C05461=1057.232,60.165,424.870,171.464,30.590,155.709
C05462=1057.237,60.415,424.853,171.466,30.593,155.709
C05463=1057.243,60.664,424.836,171.467,30.594,155.710
C05464=1057.249,60.914,424.818,171.468,30.597,155.710
C05465=1057.256,61.162,424.801,171.470,30.599,155.710
C05466=1057.263,61.412,424.784,171.472,30.602,155.711
C05467=1057.269,61.697,424.764,171.474,30.605,155.711
C05468=1057.277,61.982,424.744,171.476,30.607,155.712
C05469=1057.283,62.267,424.724,171.477,30.610,155.712
C05470=1057.291,62.551,424.705,171.479,30.613,155.712
C05471=1057.297,62.801,424.687,171.480,30.615,155.713
C05472=1057.303,63.051,424.671,171.482,30.618,155.713
C05473=1057.309,63.300,424.653,171.484,30.620,155.713
C05474=1057.316,63.550,424.635,171.485,30.622,155.714
C05475=1057.321,63.799,424.618,171.486,30.624,155.714
C05476=1057.328,64.048,424.600,171.488,30.627,155.714
C05477=1057.334,64.297,424.583,171.490,30.629,155.715
C05478=1057.341,64.547,424.565,171.491,30.632,155.715
C05479=1057.346,64.796,424.548,171.493,30.634,155.715
C05480=1057.352,65.045,424.530,171.494,30.636,155.716
C05481=1057.358,65.294,424.513,171.496,30.639,155.716
C05482=1057.365,65.544,424.495,171.497,30.641,155.717
C05483=1057.370,65.793,424.478,171.499,30.644,155.717
C05484=1057.377,66.042,424.460,171.500,30.647,155.717
C05485=1057.382,66.291,424.443,171.501,30.649,155.718
C05486=1057.389,66.541,424.425,171.503,30.651,155.718
C05487=1057.395,66.790,424.408,171.505,30.653,155.718
C05488=1057.401,67.040,424.390,171.507,30.656,155.719
C05489=1057.406,67.289,424.372,171.508,30.659,155.719
C05490=1057.413,67.538,424.355,171.509,30.661,155.720
C05491=1057.419,67.788,424.337,171.511,30.663,155.720
C05492=1057.425,68.037,424.319,171.512,30.666,155.720
C05493=1057.431,68.287,424.301,171.514,30.668,155.721
C05494=1057.437,68.535,424.284,171.516,30.671,155.721
C05495=1057.443,68.785,424.267,171.517,30.673,155.721
C05496=1057.449,69.034,424.249,171.518,30.675,155.722
C05497=1057.455,69.284,424.231,171.520,30.678,155.722
C05498=1057.461,69.533,424.214,171.522,30.680,155.722
C05499=1057.467,69.782,424.196,171.524,30.683,155.723
C05500=1057.474,70.031,424.177,171.524,30.685,155.723
C05501=1057.479,70.280,424.160,171.526,30.688,155.724
C05502=1057.486,70.530,424.142,171.528,30.690,155.724
C05503=1057.492,70.779,424.125,171.529,30.693,155.724
C05504=1057.498,71.029,424.107,171.531,30.695,155.725
C05505=1057.503,71.278,424.089,171.532,30.698,155.725
C05506=1057.510,71.527,424.072,171.534,30.700,155.726
C05507=1057.516,71.777,424.053,171.535,30.702,155.726
C05508=1057.522,72.026,424.035,171.537,30.705,155.726
C05509=1057.528,72.275,424.018,171.539,30.708,155.727
C05510=1057.534,72.524,424.000,171.540,30.710,155.727
C05511=1057.540,72.774,423.983,171.541,30.712,155.727
C05512=1057.546,73.023,423.964,171.543,30.715,155.728
C05513=1057.552,73.272,423.946,171.545,30.717,155.728
C05514=1057.558,73.522,423.928,171.546,30.720,155.728
C05515=1057.564,73.771,423.911,171.548,30.722,155.729
C05516=1057.570,74.020,423.892,171.549,30.725,155.729
C05517=1057.576,74.270,423.874,171.550,30.727,155.730
C05518=1057.582,74.519,423.857,171.552,30.730,155.730
C05519=1057.589,74.768,423.839,171.554,30.732,155.730
C05520=1057.594,75.017,423.821,171.556,30.735,155.731
C05521=1057.600,75.266,423.803,171.556,30.737,155.731
C05522=1057.607,75.516,423.785,171.558,30.739,155.731
C05523=1057.612,75.764,423.767,171.560,30.742,155.732
C05524=1057.619,76.014,423.749,171.561,30.744,155.732
C05525=1057.625,76.264,423.731,171.563,30.747,155.733
C05526=1057.630,76.512,423.713,171.564,30.749,155.733
C05527=1057.637,76.762,423.695,171.566,30.752,155.733
C05528=1057.643,77.012,423.677,171.567,30.754,155.734
C05529=1057.649,77.260,423.659,171.569,30.757,155.734
C05530=1057.655,77.510,423.641,171.571,30.759,155.734
C05531=1057.662,77.795,423.620,171.572,30.762,155.735
C05532=1057.669,78.080,423.600,171.574,30.765,155.735
C05533=1057.676,78.364,423.579,171.576,30.767,155.736
C05534=1057.683,78.649,423.558,171.578,30.771,155.736
C05535=1057.689,78.899,423.540,171.579,30.773,155.737
C05536=1057.695,79.147,423.522,171.580,30.775,155.737
C05537=1057.700,79.397,423.503,171.582,30.778,155.737
C05538=1057.706,79.647,423.485,171.584,30.781,155.738
C05539=1057.712,79.896,423.467,171.585,30.783,155.738
C05540=1057.718,80.145,423.449,171.587,30.785,155.738
C05541=1057.725,80.394,423.430,171.588,30.788,155.739
C05542=1057.730,80.643,423.413,171.589,30.791,155.739
C05543=1057.736,80.893,423.394,171.591,30.793,155.740
C05544=1057.742,81.143,423.376,171.593,30.795,155.740
C05545=1057.748,81.391,423.357,171.595,30.798,155.740
C05546=1057.754,81.641,423.339,171.596,30.801,155.741
C05547=1057.760,81.890,423.321,171.597,30.803,155.741
C05548=1057.766,82.139,423.303,171.599,30.805,155.742
C05549=1057.772,82.388,423.284,171.601,30.808,155.742
C05550=1057.778,82.638,423.265,171.602,30.811,155.742
C05551=1057.784,82.887,423.247,171.604,30.813,155.743
C05552=1057.790,83.136,423.229,171.605,30.815,155.743
C05553=1057.796,83.385,423.211,171.606,30.818,155.744
C05554=1057.802,83.635,423.193,171.608,30.821,155.744
C05555=1057.808,83.885,423.174,171.610,30.823,155.744
C05556=1057.814,84.133,423.156,171.612,30.825,155.745
C05557=1057.820,84.382,423.137,171.613,30.828,155.745
C05558=1057.826,84.632,423.119,171.614,30.830,155.745
C05559=1057.833,84.881,423.101,171.616,30.833,155.746
C05560=1057.837,85.130,423.082,171.618,30.835,155.746
C05561=1057.844,85.379,423.064,171.619,30.838,155.747
C05562=1057.850,85.629,423.045,171.621,30.840,155.747
C05563=1057.856,85.878,423.027,171.622,30.843,155.747
C05564=1057.862,86.127,423.009,171.623,30.845,155.748
C05565=1057.868,86.376,422.990,171.625,30.847,155.748
C05566=1057.874,86.626,422.972,171.627,30.850,155.748
C05567=1057.880,86.875,422.953,171.629,30.853,155.749
C05568=1057.887,87.124,422.934,171.630,30.855,155.749
C05569=1057.892,87.373,422.917,171.631,30.857,155.750
C05570=1057.898,87.623,422.898,171.633,30.860,155.750
C05571=1057.905,87.872,422.879,171.635,30.863,155.750
C05572=1057.911,88.121,422.860,171.636,30.865,155.751
C05573=1057.917,88.371,422.842,171.638,30.867,155.751
C05574=1057.923,88.619,422.824,171.639,30.870,155.752
C05575=1057.929,88.868,422.805,171.641,30.872,155.752
C05576=1057.935,89.118,422.786,171.642,30.875,155.752
C05577=1057.941,89.367,422.768,171.644,30.877,155.753
C05578=1057.948,89.616,422.750,171.646,30.880,155.753
C05579=1057.953,89.866,422.730,171.648,30.882,155.753
C05580=1057.960,90.115,422.712,171.648,30.885,155.754
C05581=1057.965,90.364,422.694,171.650,30.887,155.754
C05582=1057.972,90.613,422.675,171.652,30.890,155.754
C05583=1057.977,90.863,422.656,171.654,30.892,155.755
C05584=1057.984,91.112,422.638,171.655,30.895,155.755
C05585=1057.989,91.361,422.618,171.656,30.897,155.756
C05586=1057.996,91.610,422.600,171.658,30.900,155.756
C05587=1058.001,91.860,422.582,171.659,30.902,155.756
C05588=1058.007,92.109,422.563,171.661,30.905,155.757
C05589=1058.013,92.358,422.544,171.663,30.907,155.757
C05590=1058.019,92.607,422.525,171.665,30.910,155.758
C05591=1058.025,92.857,422.506,171.665,30.912,155.758
C05592=1058.031,93.106,422.487,171.667,30.915,155.758
C05593=1058.036,93.355,422.468,171.669,30.917,155.759
C05594=1058.043,93.604,422.450,171.671,30.920,155.759
C05595=1058.049,93.889,422.428,171.673,30.923,155.760
C05596=1058.057,94.174,422.407,171.674,30.926,155.760
C05597=1058.063,94.458,422.385,171.676,30.929,155.761
C05598=1058.070,94.743,422.363,171.678,30.931,155.761
C05599=1058.076,94.992,422.345,171.679,30.934,155.761
C05600=1058.082,95.242,422.325,171.681,30.937,155.762
C05601=1058.089,95.491,422.307,171.682,30.939,155.762
C05602=1058.094,95.740,422.288,171.684,30.941,155.763
C05603=1058.101,95.990,422.269,171.685,30.944,155.763
C05604=1058.106,96.239,422.250,171.687,30.947,155.763
C05605=1058.112,96.487,422.231,171.689,30.949,155.764
C05606=1058.118,96.737,422.212,171.691,30.951,155.764
C05607=1058.124,96.986,422.194,171.691,30.954,155.764
C05608=1058.130,97.235,422.174,171.693,30.957,155.765
C05609=1058.136,97.484,422.156,171.695,30.959,155.765
C05610=1058.142,97.734,422.136,171.697,30.961,155.766
C05611=1058.148,97.983,422.117,171.698,30.964,155.766
C05612=1058.154,98.232,422.098,171.700,30.967,155.766
C05613=1058.160,98.482,422.079,171.701,30.969,155.767
C05614=1058.166,98.731,422.061,171.703,30.971,155.767
C05615=1058.172,98.980,422.041,171.704,30.974,155.768
C05616=1058.178,99.230,422.023,171.706,30.977,155.768
C05617=1058.184,99.478,422.003,171.708,30.979,155.768
C05618=1058.191,99.728,421.984,171.710,30.981,155.769
C05619=1058.197,99.977,421.965,171.710,30.984,155.769
C05620=1058.203,100.226,421.946,171.712,30.987,155.770
C05621=1058.209,100.476,421.927,171.714,30.989,155.770
C05622=1058.215,100.725,421.908,171.716,30.991,155.770
C05623=1058.221,100.974,421.889,171.718,30.994,155.771
C05624=1058.227,101.223,421.869,171.718,30.997,155.771
C05625=1058.232,101.472,421.850,171.720,30.999,155.772
C05626=1058.239,101.721,421.831,171.722,31.002,155.772
C05627=1058.245,101.971,421.812,171.724,31.004,155.772
C05628=1058.250,102.220,421.793,171.725,31.006,155.773
C05629=1058.256,102.468,421.773,171.727,31.009,155.773
C05630=1058.262,102.718,421.754,171.728,31.012,155.773
C05631=1058.268,102.967,421.735,171.730,31.015,155.774
C05632=1058.273,103.216,421.716,171.731,31.017,155.774
C05633=1058.279,103.465,421.696,171.733,31.019,155.775
C05634=1058.285,103.715,421.677,171.735,31.022,155.775
C05635=1058.292,103.964,421.658,171.737,31.024,155.775
C05636=1058.298,104.213,421.638,171.737,31.027,155.776
C05637=1058.303,104.462,421.619,171.739,31.030,155.776
C05638=1058.309,104.711,421.600,171.741,31.032,155.777
C05639=1058.315,104.961,421.581,171.743,31.034,155.777
C05640=1058.321,105.209,421.561,171.744,31.037,155.777
C05641=1058.327,105.459,421.542,171.746,31.040,155.778
C05642=1058.333,105.708,421.523,171.747,31.042,155.778
C05643=1058.339,105.957,421.503,171.749,31.045,155.779
C05644=1058.345,106.206,421.484,171.751,31.048,155.779
C05645=1058.351,106.456,421.465,171.752,31.050,155.779
C05646=1058.357,106.704,421.445,171.754,31.052,155.780
C05647=1058.363,106.955,421.425,171.756,31.055,155.780
C05648=1058.369,107.203,421.405,171.757,31.058,155.781
C05649=1058.376,107.452,421.387,171.758,31.060,155.781
C05650=1058.381,107.702,421.367,171.760,31.062,155.781
C05651=1058.387,107.951,421.347,171.762,31.065,155.782
C05652=1058.393,108.200,421.328,171.764,31.068,155.782
C05653=1058.399,108.449,421.308,171.765,31.070,155.783
C05654=1058.405,108.698,421.289,171.766,31.073,155.783
C05655=1058.411,108.947,421.270,171.768,31.075,155.783
C05656=1058.417,109.196,421.250,171.770,31.077,155.784
C05657=1058.423,109.446,421.231,171.772,31.080,155.784
C05658=1058.429,109.695,421.211,171.773,31.083,155.785
C05659=1058.436,109.980,421.189,171.775,31.085,155.785
C05660=1058.443,110.264,421.166,171.777,31.088,155.785
C05661=1058.450,110.550,421.144,171.779,31.091,155.786
C05662=1058.457,110.835,421.122,171.781,31.094,155.786
C05663=1058.463,111.083,421.102,171.782,31.097,155.787
C05664=1058.469,111.333,421.083,171.784,31.099,155.787
C05665=1058.475,111.582,421.063,171.785,31.102,155.788
C05666=1058.481,111.830,421.043,171.787,31.104,155.788
C05667=1058.486,112.080,421.024,171.789,31.107,155.788
C05668=1058.492,112.329,421.004,171.790,31.109,155.789
C05669=1058.498,112.578,420.985,171.792,31.112,155.789
C05670=1058.505,112.828,420.964,171.794,31.115,155.790
C05671=1058.510,113.077,420.945,171.795,31.117,155.790
C05672=1058.516,113.326,420.925,171.797,31.119,155.790
C05673=1058.522,113.575,420.905,171.798,31.122,155.791
C05674=1058.528,113.824,420.886,171.800,31.124,155.791
C05675=1058.534,114.073,420.866,171.802,31.127,155.791
C05676=1058.540,114.322,420.846,171.804,31.130,155.792
C05677=1058.546,114.571,420.827,171.805,31.132,155.792
C05678=1058.551,114.821,420.806,171.806,31.135,155.793
C05679=1058.557,115.070,420.786,171.808,31.138,155.793
C05680=1058.563,115.319,420.767,171.810,31.140,155.794
C05681=1058.569,115.568,420.747,171.812,31.143,155.794
C05682=1058.575,115.817,420.727,171.814,31.146,155.794
C05683=1058.580,116.067,420.707,171.814,31.148,155.795
C05684=1058.586,116.315,420.687,171.816,31.151,155.795
C05685=1058.592,116.564,420.667,171.818,31.153,155.796
C05686=1058.598,116.813,420.647,171.820,31.156,155.796
C05687=1058.604,117.064,420.627,171.822,31.158,155.796
C05688=1058.610,117.312,420.607,171.823,31.161,155.797
C05689=1058.616,117.561,420.587,171.824,31.163,155.797
C05690=1058.622,117.810,420.567,171.826,31.166,155.798
C05691=1058.627,118.059,420.548,171.828,31.169,155.798
C05692=1058.633,118.309,420.527,171.830,31.171,155.798
C05693=1058.639,118.558,420.507,171.831,31.174,155.799
C05694=1058.645,118.807,420.487,171.833,31.177,155.799
C05695=1058.651,119.056,420.467,171.834,31.179,155.800
C05696=1058.656,119.305,420.447,171.836,31.182,155.800
C05697=1058.662,119.554,420.427,171.838,31.185,155.801
C05698=1058.668,119.803,420.407,171.839,31.187,155.801
C05699=1058.675,120.053,420.387,171.841,31.190,155.801
C05700=1058.680,120.302,420.366,171.843,31.192,155.802
C05701=1058.686,120.551,420.346,171.844,31.194,155.802
C05702=1058.692,120.799,420.326,171.846,31.197,155.803
C05703=1058.698,121.049,420.307,171.847,31.200,155.803
C05704=1058.703,121.299,420.286,171.849,31.202,155.803
C05705=1058.709,121.547,420.266,171.851,31.205,155.804
C05706=1058.715,121.796,420.246,171.853,31.208,155.804
C05707=1058.721,122.045,420.226,171.854,31.210,155.805
C05708=1058.727,122.295,420.205,171.856,31.213,155.805
C05709=1058.733,122.544,420.185,171.857,31.215,155.805
C05710=1058.739,122.792,420.165,171.859,31.218,155.806
C05711=1058.745,123.042,420.145,171.861,31.220,155.806
C05712=1058.751,123.291,420.124,171.863,31.223,155.807
C05713=1058.757,123.540,420.105,171.865,31.225,155.807
C05714=1058.763,123.789,420.085,171.866,31.228,155.807
C05715=1058.769,124.039,420.064,171.867,31.231,155.808
C05716=1058.775,124.287,420.044,171.869,31.233,155.808
C05717=1058.781,124.536,420.024,171.871,31.236,155.809
C05718=1058.786,124.785,420.003,171.873,31.239,155.809
C05719=1058.793,125.035,419.983,171.875,31.241,155.810
C05720=1058.799,125.284,419.963,171.876,31.243,155.810
C05721=1058.804,125.533,419.942,171.877,31.246,155.810
C05722=1058.811,125.782,419.922,171.879,31.248,155.811
C05723=1058.817,126.067,419.899,171.881,31.252,155.811
C05724=1058.824,126.351,419.876,171.884,31.255,155.812
C05725=1058.831,126.636,419.853,171.886,31.257,155.812
C05726=1058.838,126.921,419.829,171.887,31.260,155.813
C05727=1058.844,127.170,419.809,171.889,31.263,155.813
C05728=1058.850,127.419,419.789,171.890,31.266,155.813
C05729=1058.855,127.669,419.768,171.892,31.268,155.814
C05730=1058.862,127.917,419.748,171.894,31.270,155.814
C05731=1058.868,128.167,419.727,171.896,31.273,155.815
C05732=1058.874,128.415,419.707,171.897,31.276,155.815
C05733=1058.880,128.664,419.687,171.899,31.278,155.815
C05734=1058.886,128.914,419.666,171.901,31.281,155.816
C05735=1058.891,129.163,419.646,171.903,31.284,155.816
C05736=1058.897,129.412,419.626,171.904,31.285,155.817
C05737=1058.904,129.661,419.605,171.906,31.288,155.817
C05738=1058.910,129.910,419.584,171.908,31.291,155.817
C05739=1058.916,130.159,419.564,171.909,31.293,155.818
C05740=1058.922,130.408,419.544,171.911,31.296,155.818
C05741=1058.928,130.658,419.523,171.913,31.299,155.819
C05742=1058.934,130.906,419.502,171.915,31.301,155.819
C05743=1058.940,131.155,419.482,171.917,31.303,155.819
C05744=1058.946,131.405,419.462,171.918,31.306,155.820
C05745=1058.952,131.654,419.442,171.920,31.309,155.820
C05746=1058.958,131.903,419.420,171.921,31.311,155.821
C05747=1058.964,132.152,419.400,171.923,31.314,155.821
C05748=1058.970,132.401,419.379,171.925,31.317,155.821
C05749=1058.976,132.650,419.359,171.927,31.319,155.822
C05750=1058.982,132.899,419.338,171.929,31.322,155.822
C05751=1058.988,133.149,419.317,171.930,31.324,155.823
C05752=1058.994,133.398,419.297,171.931,31.327,155.823
C05753=1058.999,133.646,419.276,171.933,31.330,155.824
C05754=1059.005,133.896,419.255,171.935,31.332,155.824
C05755=1059.011,134.144,419.234,171.937,31.335,155.824
C05756=1059.017,134.394,419.213,171.939,31.338,155.825
C05757=1059.023,134.643,419.193,171.941,31.340,155.825
C05758=1059.029,134.891,419.172,171.943,31.343,155.826
C05759=1059.035,135.141,419.151,171.944,31.346,155.826
C05760=1059.041,135.390,419.131,171.945,31.348,155.826
C05761=1059.047,135.639,419.109,171.947,31.351,155.827
C05762=1059.052,135.888,419.089,171.949,31.353,155.827
C05763=1059.059,136.137,419.068,171.951,31.356,155.828
C05764=1059.064,136.386,419.047,171.953,31.358,155.828
C05765=1059.070,136.635,419.026,171.954,31.361,155.828
C05766=1059.076,136.884,419.006,171.956,31.363,155.829
C05767=1059.082,137.133,418.984,171.958,31.366,155.829
C05768=1059.088,137.382,418.964,171.960,31.369,155.830
C05769=1059.094,137.631,418.943,171.961,31.371,155.830
C05770=1059.100,137.881,418.922,171.963,31.374,155.831
C05771=1059.105,138.129,418.901,171.965,31.376,155.831
C05772=1059.112,138.379,418.880,171.966,31.379,155.831
C05773=1059.118,138.627,418.859,171.968,31.382,155.832
C05774=1059.123,138.877,418.838,171.970,31.384,155.832
C05775=1059.129,139.125,418.817,171.972,31.387,155.833
C05776=1059.136,139.375,418.797,171.974,31.390,155.833
C05777=1059.141,139.623,418.775,171.976,31.392,155.833
C05778=1059.147,139.873,418.754,171.978,31.395,155.834
C05779=1059.153,140.121,418.734,171.979,31.398,155.834
C05780=1059.160,140.371,418.712,171.980,31.400,155.835
C05781=1059.165,140.620,418.691,171.982,31.403,155.835
C05782=1059.171,140.869,418.670,171.984,31.405,155.836
C05783=1059.176,141.118,418.649,171.986,31.408,155.836
C05784=1059.182,141.367,418.628,171.988,31.411,155.836
C05785=1059.188,141.616,418.606,171.990,31.413,155.837
C05786=1059.194,141.866,418.585,171.991,31.416,155.837
C05787=1059.200,142.150,418.561,171.993,31.419,155.838
C05788=1059.208,142.434,418.537,171.995,31.422,155.838
C05789=1059.215,142.719,418.513,171.997,31.425,155.839
C05790=1059.221,143.004,418.489,172.000,31.428,155.839
C05791=1059.226,143.253,418.468,172.002,31.431,155.840
C05792=1059.233,143.502,418.446,172.003,31.434,155.840
C05793=1059.239,143.750,418.425,172.004,31.436,155.841
C05794=1059.245,144.000,418.404,172.006,31.439,155.841
C05795=1059.250,144.248,418.383,172.008,31.441,155.841
C05796=1059.256,144.498,418.361,172.010,31.444,155.842
C05797=1059.262,144.746,418.340,172.012,31.447,155.842
C05798=1059.268,144.996,418.319,172.014,31.449,155.843
C05799=1059.274,145.233,418.298,172.015,31.452,155.843
C05800=1059.279,145.470,418.279,172.017,31.455,155.843
C05801=1059.285,145.707,418.258,172.019,31.457,155.844
C05802=1059.290,145.944,418.238,172.021,31.459,155.844
C05803=1059.296,146.181,418.217,172.022,31.462,155.845
C05804=1059.302,146.418,418.198,172.024,31.464,155.845
C05805=1059.308,146.655,418.177,172.026,31.467,155.845
C05806=1059.313,146.892,418.157,172.027,31.470,155.846
C05807=1059.319,147.141,418.135,172.029,31.472,155.846
C05808=1059.325,147.391,418.114,172.031,31.475,155.847
C05809=1059.331,147.639,418.093,172.033,31.478,155.847
C05810=1059.337,147.888,418.071,172.035,31.480,155.848
C05811=1059.342,148.137,418.050,172.037,31.483,155.848
C05812=1059.348,148.386,418.028,172.039,31.485,155.848
C05813=1059.355,148.635,418.006,172.040,31.488,155.849
C05814=1059.360,148.884,417.985,172.042,31.491,155.849
C05815=1059.366,149.134,417.964,172.044,31.493,155.850
C05816=1059.372,149.382,417.943,172.045,31.496,155.850
C05817=1059.378,149.631,417.921,172.047,31.498,155.851
C05818=1059.384,149.881,417.900,172.049,31.501,155.851
C05819=1059.390,150.129,417.878,172.051,31.504,155.851
C05820=1059.396,150.378,417.857,172.052,31.506,155.852
C05821=1059.401,150.628,417.834,172.054,31.510,155.852
C05822=1059.407,150.876,417.813,172.056,31.512,155.853
C05823=1059.413,151.125,417.792,172.058,31.515,155.853
C05824=1059.419,151.375,417.770,172.060,31.517,155.854
C05825=1059.425,151.623,417.749,172.062,31.520,155.854
C05826=1059.431,151.872,417.727,172.064,31.523,155.854
C05827=1059.436,152.122,417.705,172.065,31.525,155.855
C05828=1059.442,152.370,417.683,172.067,31.528,155.855
C05829=1059.448,152.619,417.661,172.069,31.531,155.856
C05830=1059.454,152.868,417.640,172.071,31.533,155.856
C05831=1059.460,153.117,417.618,172.073,31.536,155.857
C05832=1059.466,153.366,417.597,172.075,31.539,155.857
C05833=1059.471,153.615,417.574,172.077,31.542,155.857
C05834=1059.477,153.864,417.553,172.078,31.544,155.858
C05835=1059.483,154.113,417.532,172.080,31.547,155.858
C05836=1059.489,154.362,417.510,172.082,31.550,155.859
C05837=1059.496,154.612,417.488,172.084,31.552,155.859
C05838=1059.501,154.860,417.466,172.086,31.555,155.860
C05839=1059.507,155.109,417.444,172.088,31.558,155.860
C05840=1059.513,155.358,417.422,172.090,31.560,155.860
C05841=1059.519,155.607,417.401,172.092,31.563,155.861
C05842=1059.524,155.856,417.379,172.093,31.566,155.861
C05843=1059.530,156.105,417.357,172.095,31.569,155.862
C05844=1059.537,156.354,417.335,172.097,31.571,155.862
C05845=1059.541,156.603,417.313,172.099,31.574,155.863
C05846=1059.548,156.852,417.291,172.101,31.576,155.863
C05847=1059.554,157.101,417.270,172.103,31.580,155.864
C05848=1059.560,157.350,417.247,172.105,31.582,155.864
C05849=1059.565,157.599,417.226,172.106,31.585,155.864
C05850=1059.571,157.848,417.204,172.108,31.588,155.865
C05851=1059.579,158.156,417.176,172.111,31.591,155.865
C05852=1059.586,158.464,417.149,172.113,31.594,155.866
C05853=1059.593,158.772,417.123,172.116,31.597,155.866
C05854=1059.600,159.081,417.095,172.118,31.601,155.867
C05855=1059.606,159.330,417.073,172.119,31.604,155.868
C05856=1059.613,159.579,417.051,172.121,31.607,155.868
C05857=1059.617,159.828,417.029,172.123,31.609,155.868
C05858=1059.624,160.076,417.007,172.125,31.612,155.869
C05859=1059.630,160.325,416.985,172.127,31.614,155.869
C05860=1059.636,160.574,416.962,172.129,31.617,155.870
C05861=1059.642,160.824,416.940,172.131,31.620,155.870
C05862=1059.647,161.073,416.918,172.133,31.623,155.871
C05863=1059.653,161.321,416.896,172.134,31.625,155.871
C05864=1059.659,161.570,416.874,172.136,31.628,155.871
C05865=1059.664,161.819,416.851,172.138,31.631,155.872
C05866=1059.670,162.068,416.830,172.140,31.634,155.872
C05867=1059.676,162.317,416.807,172.142,31.637,155.873
C05868=1059.681,162.566,416.785,172.144,31.640,155.873
C05869=1059.688,162.815,416.762,172.146,31.642,155.874
C05870=1059.693,163.064,416.740,172.147,31.645,155.874
C05871=1059.698,163.313,416.717,172.150,31.648,155.875
C05872=1059.704,163.562,416.696,172.152,31.651,155.875
C05873=1059.710,163.811,416.673,172.154,31.654,155.876
C05874=1059.715,164.060,416.651,172.156,31.657,155.876
C05875=1059.721,164.308,416.628,172.158,31.659,155.877
C05876=1059.727,164.557,416.606,172.160,31.662,155.877
C05877=1059.732,164.806,416.584,172.162,31.665,155.877
C05878=1059.738,165.055,416.561,172.163,31.668,155.878
C05879=1059.744,165.305,416.539,172.165,31.670,155.878
C05880=1059.750,165.553,416.516,172.167,31.674,155.879
C05881=1059.755,165.802,416.493,172.169,31.676,155.879
C05882=1059.761,166.051,416.471,172.171,31.679,155.880
C05883=1059.767,166.300,416.449,172.173,31.682,155.880
C05884=1059.773,166.549,416.427,172.175,31.685,155.881
C05885=1059.778,166.798,416.404,172.176,31.687,155.881
C05886=1059.785,167.047,416.381,172.178,31.690,155.882
C05887=1059.790,167.296,416.359,172.180,31.693,155.882
C05888=1059.795,167.544,416.336,172.182,31.696,155.883
C05889=1059.801,167.793,416.314,172.184,31.699,155.883
C05890=1059.808,168.042,416.291,172.187,31.702,155.883
C05891=1059.813,168.291,416.269,172.189,31.704,155.884
C05892=1059.819,168.540,416.246,172.191,31.707,155.884
C05893=1059.824,168.789,416.223,172.192,31.710,155.885
C05894=1059.831,169.038,416.201,172.194,31.713,155.885
C05895=1059.836,169.287,416.178,172.196,31.716,155.886
C05896=1059.841,169.536,416.156,172.198,31.719,155.886
C05897=1059.847,169.784,416.133,172.200,31.721,155.887
C05898=1059.853,170.033,416.110,172.202,31.724,155.887
C05899=1059.859,170.283,416.088,172.204,31.727,155.888
C05900=1059.865,170.531,416.065,172.206,31.730,155.888
C05901=1059.871,170.780,416.042,172.207,31.733,155.889
C05902=1059.876,171.029,416.020,172.210,31.735,155.889
C05903=1059.883,171.278,415.997,172.212,31.738,155.889
C05904=1059.888,171.527,415.974,172.214,31.741,155.890
C05905=1059.894,171.776,415.952,172.216,31.744,155.890
C05906=1059.900,172.025,415.929,172.218,31.747,155.891
C05907=1059.905,172.274,415.906,172.220,31.750,155.891
C05908=1059.912,172.523,415.884,172.222,31.752,155.892
C05909=1059.918,172.772,415.861,172.223,31.755,155.892
C05910=1059.923,173.020,415.838,172.225,31.758,155.893
C05911=1059.929,173.269,415.815,172.228,31.761,155.893
C05912=1059.935,173.518,415.792,172.230,31.763,155.894
C05913=1059.941,173.767,415.770,172.232,31.767,155.894
C05914=1059.947,174.016,415.747,172.234,31.769,155.895
C05915=1059.954,174.300,415.721,172.236,31.772,155.895
C05916=1059.960,174.584,415.694,172.238,31.776,155.896
C05917=1059.967,174.868,415.669,172.240,31.779,155.896
C05918=1059.973,175.151,415.643,172.243,31.782,155.897
C05919=1059.979,175.401,415.619,172.245,31.785,155.897
C05920=1059.985,175.650,415.596,172.247,31.788,155.898
C05921=1059.992,175.898,415.574,172.249,31.791,155.898
C05922=1059.997,176.147,415.551,172.251,31.793,155.898
C05923=1060.003,176.396,415.528,172.253,31.796,155.899
C05924=1060.009,176.645,415.505,172.255,31.799,155.899
C05925=1060.015,176.894,415.482,172.257,31.802,155.900
C05926=1060.020,177.143,415.459,172.259,31.804,155.900
C05927=1060.027,177.391,415.437,172.261,31.808,155.901
C05928=1060.033,177.640,415.414,172.263,31.810,155.901
C05929=1060.038,177.889,415.391,172.265,31.813,155.902
C05930=1060.045,178.139,415.368,172.268,31.816,155.902
C05931=1060.050,178.388,415.345,172.270,31.819,155.903
C05932=1060.056,178.636,415.321,172.271,31.821,155.903
C05933=1060.062,178.885,415.298,172.273,31.825,155.904
C05934=1060.069,179.133,415.276,172.275,31.827,155.904
C05935=1060.074,179.382,415.253,172.277,31.830,155.904
C05936=1060.080,179.631,415.230,172.280,31.833,155.905
C05937=1060.086,179.881,415.207,172.282,31.836,155.905
C05938=1060.092,180.130,415.184,172.284,31.838,155.906
C05939=1060.098,180.378,415.160,172.286,31.841,155.906
C05940=1060.104,180.627,415.137,172.288,31.844,155.907
C05941=1060.110,180.876,415.114,172.290,31.847,155.907
C05942=1060.115,181.125,415.091,172.292,31.850,155.908
C05943=1060.123,181.373,415.068,172.294,31.853,155.908
C05944=1060.128,181.622,415.045,172.296,31.855,155.909
C05945=1060.134,181.871,415.022,172.298,31.858,155.909
C05946=1060.140,182.120,414.999,172.301,31.861,155.910
C05947=1060.146,182.368,414.975,172.303,31.864,155.910
C05948=1060.152,182.618,414.952,172.305,31.867,155.911
C05949=1060.158,182.867,414.929,172.306,31.869,155.911
C05950=1060.164,183.116,414.906,172.308,31.872,155.911
C05951=1060.170,183.364,414.882,172.311,31.875,155.912
C05952=1060.176,183.614,414.859,172.313,31.878,155.912
C05953=1060.183,183.862,414.837,172.315,31.881,155.913
C05954=1060.189,184.110,414.813,172.317,31.884,155.913
C05955=1060.194,184.359,414.790,172.320,31.886,155.914
C05956=1060.200,184.609,414.766,172.322,31.890,155.914
C05957=1060.206,184.857,414.743,172.324,31.892,155.915
C05958=1060.212,185.106,414.720,172.325,31.895,155.915
C05959=1060.217,185.355,414.695,172.327,31.898,155.916
C05960=1060.223,185.604,414.672,172.330,31.901,155.916
C05961=1060.229,185.852,414.649,172.332,31.905,155.917
C05962=1060.234,186.102,414.625,172.334,31.907,155.917
C05963=1060.240,186.350,414.601,172.336,31.910,155.918
C05964=1060.245,186.600,414.578,172.338,31.913,155.918
C05965=1060.251,186.848,414.554,172.341,31.916,155.919
C05966=1060.257,187.097,414.531,172.342,31.919,155.919
C05967=1060.262,187.345,414.507,172.344,31.923,155.920
C05968=1060.269,187.594,414.483,172.346,31.925,155.920
C05969=1060.274,187.843,414.459,172.348,31.928,155.921
C05970=1060.280,188.092,414.436,172.351,31.931,155.921
C05971=1060.286,188.341,414.413,172.353,31.934,155.922
C05972=1060.291,188.589,414.388,172.355,31.937,155.922
C05973=1060.297,188.839,414.365,172.357,31.940,155.923
C05974=1060.303,189.087,414.341,172.360,31.943,155.923
C05975=1060.309,189.336,414.317,172.361,31.946,155.924
C05976=1060.314,189.585,414.294,172.363,31.949,155.924
C05977=1060.320,189.834,414.270,172.365,31.952,155.925
C05978=1060.326,190.082,414.246,172.368,31.956,155.925
C05979=1060.333,190.366,414.219,172.370,31.959,155.926
C05980=1060.339,190.649,414.192,172.373,31.962,155.926
C05981=1060.346,190.933,414.165,172.375,31.966,155.927
C05982=1060.353,191.216,414.137,172.378,31.969,155.928
C05983=1060.358,191.465,414.113,172.379,31.972,155.928
C05984=1060.364,191.714,414.090,172.381,31.975,155.928
C05985=1060.369,191.962,414.066,172.384,31.978,155.929
C05986=1060.376,192.211,414.042,172.386,31.981,155.929
C05987=1060.381,192.460,414.018,172.388,31.984,155.930
C05988=1060.387,192.709,413.995,172.390,31.987,155.931
C05989=1060.393,192.958,413.970,172.393,31.990,155.931
C05990=1060.399,193.207,413.947,172.395,31.993,155.932
C05991=1060.404,193.455,413.922,172.397,31.996,155.932
C05992=1060.411,193.705,413.899,172.399,31.999,155.932
C05993=1060.416,193.953,413.875,172.401,32.002,155.933
C05994=1060.423,194.202,413.851,172.403,32.005,155.934
C05995=1060.429,194.451,413.827,172.405,32.008,155.934
C05996=1060.434,194.699,413.803,172.408,32.011,155.935
C05997=1060.441,194.948,413.779,172.410,32.014,155.935
C05998=1060.446,195.197,413.754,172.412,32.017,155.935
C05999=1060.452,195.446,413.732,172.415,32.020,155.936
C06000=1060.457,195.695,413.707,172.417,32.023,155.937
C06001=1060.463,195.943,413.683,172.418,32.026,155.937
C06002=1060.469,196.192,413.659,172.421,32.029,155.938
C06003=1060.475,196.441,413.635,172.423,32.032,155.938
C06004=1060.481,196.689,413.611,172.425,32.035,155.939
C06005=1060.487,196.938,413.587,172.428,32.038,155.939
C06006=1060.493,197.187,413.562,172.430,32.041,155.940
C06007=1060.499,197.436,413.538,172.432,32.044,155.940
C06008=1060.505,197.684,413.514,172.435,32.047,155.941
C06009=1060.511,197.933,413.490,172.437,32.050,155.941
C06010=1060.517,198.182,413.466,172.439,32.053,155.942
C06011=1060.522,198.431,413.441,172.441,32.056,155.942
C06012=1060.528,198.680,413.418,172.443,32.059,155.943
C06013=1060.534,198.929,413.393,172.445,32.063,155.943
C06014=1060.540,199.177,413.369,172.448,32.066,155.944
C06015=1060.546,199.426,413.345,172.450,32.068,155.944
C06016=1060.552,199.675,413.321,172.452,32.072,155.945
C06017=1060.558,199.924,413.296,172.455,32.075,155.945
C06018=1060.564,200.172,413.273,172.457,32.077,155.946
C06019=1060.570,200.421,413.247,172.459,32.081,155.946
C06020=1060.577,200.669,413.224,172.461,32.084,155.947
C06021=1060.582,200.919,413.199,172.463,32.087,155.947
C06022=1060.588,201.167,413.175,172.465,32.090,155.948
C06023=1060.594,201.416,413.151,172.468,32.093,155.948
C06024=1060.600,201.665,413.127,172.470,32.096,155.949
C06025=1060.606,201.914,413.103,172.472,32.099,155.949
C06026=1060.612,202.162,413.078,172.475,32.102,155.950
C06027=1060.618,202.411,413.053,172.477,32.105,155.950
C06028=1060.623,202.659,413.029,172.480,32.108,155.951
C06029=1060.630,202.908,413.005,172.482,32.111,155.951
C06030=1060.635,203.156,412.980,172.483,32.115,155.952
C06031=1060.641,203.406,412.955,172.486,32.118,155.952
C06032=1060.647,203.654,412.931,172.488,32.121,155.953
C06033=1060.652,203.904,412.906,172.490,32.124,155.954
C06034=1060.658,204.152,412.881,172.493,32.127,155.954
C06035=1060.665,204.401,412.857,172.495,32.130,155.955
C06036=1060.671,204.650,412.833,172.498,32.133,155.955
C06037=1060.676,204.898,412.808,172.500,32.136,155.956
C06038=1060.682,205.147,412.783,172.502,32.140,155.956
C06039=1060.687,205.396,412.759,172.505,32.143,155.957
C06040=1060.694,205.644,412.733,172.506,32.146,155.957
C06041=1060.699,205.893,412.709,172.508,32.149,155.958
C06042=1060.705,206.142,412.684,172.511,32.153,155.958
C06043=1060.730,207.190,412.580,172.690,32.237,155.967
C06044=1060.736,207.419,412.557,172.692,32.241,155.968
C06045=1060.741,207.648,412.534,172.694,32.245,155.969
C06046=1060.747,207.877,412.510,172.696,32.248,155.969
C06047=1060.752,208.106,412.486,172.696,32.252,155.970
C06048=1060.758,208.335,412.463,172.698,32.255,155.971
C06049=1060.764,208.564,412.439,172.700,32.259,155.971
C06050=1060.770,208.793,412.416,172.702,32.263,155.972
C06051=1060.775,209.022,412.392,172.704,32.267,155.973
C06052=1060.782,209.270,412.367,172.706,32.271,155.974
C06053=1060.787,209.519,412.341,172.708,32.275,155.974
C06054=1060.793,209.767,412.315,172.710,32.279,155.975
C06055=1060.800,210.016,412.289,172.712,32.283,155.976
C06056=1060.806,210.265,412.264,172.714,32.287,155.976
C06057=1060.811,210.514,412.238,172.716,32.291,155.977
C06058=1060.818,210.762,412.212,172.717,32.295,155.978
C06059=1060.824,211.011,412.187,172.719,32.299,155.979
C06060=1060.830,211.260,412.160,172.721,32.303,155.979
C06061=1060.837,211.508,412.134,172.723,32.306,155.980
C06062=1060.843,211.757,412.109,172.725,32.311,155.981
C06063=1060.848,212.006,412.083,172.727,32.314,155.982
C06064=1060.855,212.254,412.057,172.729,32.319,155.982
C06065=1060.861,212.503,412.032,172.732,32.323,155.983
C06066=1060.867,212.752,412.006,172.734,32.327,155.984
C06067=1060.873,213.000,411.980,172.736,32.331,155.985
C06068=1060.879,213.248,411.954,172.738,32.335,155.985
C06069=1060.885,213.497,411.928,172.740,32.339,155.986
C06070=1060.891,213.745,411.902,172.741,32.343,155.987
C06071=1060.897,213.994,411.876,172.743,32.347,155.988
C06072=1060.903,214.242,411.850,172.745,32.351,155.988
C06073=1060.909,214.491,411.825,172.747,32.355,155.989
C06074=1060.916,214.740,411.798,172.749,32.359,155.990
C06075=1060.921,214.989,411.772,172.751,32.363,155.991
C06076=1060.928,215.237,411.746,172.753,32.367,155.991
C06077=1060.934,215.485,411.719,172.755,32.371,155.992
C06078=1060.940,215.734,411.694,172.758,32.375,155.993
C06079=1060.946,215.983,411.667,172.760,32.379,155.993
C06080=1060.952,216.231,411.642,172.762,32.383,155.994
C06081=1060.957,216.480,411.615,172.764,32.387,155.995
C06082=1060.964,216.729,411.590,172.766,32.391,155.996
C06083=1060.970,216.977,411.563,172.767,32.395,155.996
C06084=1060.976,217.226,411.538,172.769,32.399,155.997
C06085=1060.982,217.474,411.511,172.771,32.403,155.998
C06086=1060.989,217.722,411.485,172.773,32.407,155.999
C06087=1060.994,217.971,411.459,172.775,32.411,155.999
C06088=1061.001,218.220,411.433,172.778,32.415,156.000
C06089=1061.007,218.468,411.406,172.780,32.419,156.001
C06090=1061.013,218.717,411.381,172.782,32.423,156.002
C06091=1061.019,218.965,411.354,172.784,32.426,156.002
C06092=1061.025,219.214,411.328,172.786,32.431,156.003
C06093=1061.031,219.463,411.302,172.788,32.434,156.004
C06094=1061.038,219.711,411.276,172.790,32.438,156.004
C06095=1061.044,219.960,411.249,172.792,32.442,156.005
C06096=1061.050,220.208,411.224,172.795,32.446,156.006
C06097=1061.056,220.457,411.197,172.796,32.450,156.007
C06098=1061.062,220.706,411.170,172.798,32.454,156.007
C06099=1061.069,220.954,411.144,172.800,32.458,156.008
C06100=1061.075,221.185,411.120,172.802,32.462,156.009
C06101=1061.080,221.417,411.095,172.804,32.466,156.009
C06102=1061.085,221.648,411.070,172.806,32.469,156.010
C06103=1061.091,221.880,411.046,172.808,32.473,156.011
C06104=1061.097,222.112,411.021,172.810,32.477,156.011
C06105=1061.103,222.343,410.997,172.812,32.480,156.012
C06106=1061.108,222.574,410.971,172.814,32.484,156.013
C06107=1061.113,222.805,410.947,172.816,32.488,156.014
C06108=1061.120,223.053,410.921,172.818,32.491,156.014
C06109=1061.126,223.303,410.894,172.820,32.496,156.015
C06110=1061.132,223.551,410.868,172.822,32.499,156.016
C06111=1061.137,223.800,410.841,172.824,32.503,156.016
C06112=1061.144,224.048,410.815,172.827,32.507,156.017
C06113=1061.150,224.297,410.788,172.829,32.512,156.018
C06114=1061.156,224.545,410.761,172.830,32.515,156.019
C06115=1061.162,224.794,410.735,172.832,32.519,156.019
C06116=1061.168,225.042,410.708,172.834,32.523,156.020
C06117=1061.175,225.291,410.682,172.836,32.527,156.021
C06118=1061.181,225.539,410.655,172.839,32.531,156.022
C06119=1061.186,225.788,410.628,172.841,32.535,156.022
C06120=1061.193,226.037,410.601,172.843,32.539,156.023
C06121=1061.198,226.285,410.575,172.845,32.543,156.024
C06122=1061.205,226.533,410.549,172.847,32.546,156.024
C06123=1061.211,226.782,410.522,172.850,32.551,156.025
C06124=1061.217,227.030,410.495,172.852,32.554,156.026
C06125=1061.223,227.279,410.468,172.854,32.558,156.027
C06126=1061.230,227.527,410.441,172.856,32.562,156.027
C06127=1061.235,227.776,410.414,172.858,32.566,156.028
C06128=1061.242,228.024,410.388,172.861,32.570,156.029
C06129=1061.248,228.273,410.361,172.863,32.574,156.030
C06130=1061.254,228.521,410.334,172.865,32.578,156.030
C06131=1061.260,228.770,410.307,172.867,32.581,156.031
C06132=1061.266,229.018,410.281,172.869,32.586,156.032
C06133=1061.273,229.268,410.254,172.871,32.589,156.032
C06134=1061.279,229.515,410.227,172.873,32.593,156.033
C06135=1061.285,229.763,410.200,172.875,32.597,156.034
C06136=1061.291,230.013,410.173,172.877,32.601,156.035
C06137=1061.297,230.261,410.146,172.879,32.605,156.035
C06138=1061.303,230.509,410.118,172.882,32.609,156.036
C06139=1061.309,230.758,410.091,172.884,32.613,156.037
C06140=1061.315,231.006,410.065,172.886,32.617,156.038
C06141=1061.321,231.255,410.038,172.888,32.621,156.038
C06142=1061.327,231.503,410.010,172.891,32.625,156.039
C06143=1061.334,231.752,409.983,172.893,32.629,156.040
C06144=1061.339,232.000,409.957,172.895,32.633,156.040
C06145=1061.345,232.248,409.929,172.897,32.637,156.041
C06146=1061.352,232.497,409.902,172.900,32.640,156.042
C06147=1061.358,232.746,409.876,172.902,32.645,156.043
C06148=1061.364,232.994,409.848,172.904,32.648,156.043
C06149=1061.370,233.242,409.821,172.906,32.652,156.044
C06150=1061.376,233.491,409.794,172.908,32.656,156.045
C06151=1061.382,233.739,409.766,172.911,32.660,156.045
C06152=1061.388,233.989,409.739,172.913,32.664,156.046
C06153=1061.394,234.236,409.712,172.915,32.668,156.047
C06154=1061.401,234.485,409.685,172.917,32.672,156.048
C06155=1061.407,234.733,409.658,172.920,32.676,156.048
C06156=1061.412,234.960,409.632,172.921,32.680,156.049
C06157=1061.418,235.189,409.608,172.923,32.683,156.050
C06158=1061.423,235.416,409.583,172.925,32.686,156.050
C06159=1061.429,235.644,409.557,172.927,32.690,156.051
C06160=1061.434,235.871,409.533,172.929,32.694,156.052
C06161=1061.439,236.098,409.508,172.931,32.697,156.052
C06162=1061.446,236.326,409.483,172.933,32.701,156.053
C06163=1061.451,236.553,409.457,172.935,32.705,156.054
C06164=1061.457,236.802,409.430,172.938,32.708,156.054
C06165=1061.463,237.050,409.403,172.940,32.712,156.055
C06166=1061.469,237.299,409.375,172.942,32.716,156.056
C06167=1061.475,237.547,409.348,172.944,32.720,156.057
C06168=1061.482,237.795,409.320,172.947,32.724,156.057
C06169=1061.487,238.043,409.294,172.949,32.728,156.058
C06170=1061.494,238.292,409.266,172.951,32.732,156.059
C06171=1061.500,238.541,409.238,172.954,32.735,156.059
C06172=1061.506,238.789,409.211,172.956,32.740,156.060
C06173=1061.513,239.037,409.183,172.958,32.743,156.061
C06174=1061.519,239.285,409.156,172.961,32.747,156.062
C06175=1061.524,239.535,409.128,172.963,32.751,156.062
C06176=1061.530,239.782,409.101,172.965,32.755,156.063
C06177=1061.537,240.031,409.073,172.967,32.758,156.064
C06178=1061.543,240.280,409.046,172.970,32.763,156.065
C06179=1061.549,240.528,409.018,172.972,32.766,156.065
C06180=1061.555,240.776,408.991,172.974,32.770,156.066
C06181=1061.561,241.025,408.962,172.977,32.774,156.067
C06182=1061.567,241.273,408.935,172.979,32.778,156.067
C06183=1061.574,241.522,408.908,172.981,32.782,156.068
C06184=1061.579,241.770,408.880,172.984,32.786,156.069
C06185=1061.586,242.018,408.852,172.986,32.790,156.070
C06186=1061.592,242.267,408.824,172.988,32.793,156.070
C06187=1061.598,242.515,408.796,172.991,32.797,156.071
C06188=1061.605,242.763,408.769,172.993,32.801,156.072
C06189=1061.610,243.013,408.741,172.995,32.805,156.073
C06190=1061.616,243.260,408.714,172.998,32.809,156.073
C06191=1061.622,243.509,408.685,173.000,32.813,156.074
C06192=1061.628,243.757,408.658,173.002,32.817,156.075
C06193=1061.634,244.006,408.630,173.004,32.821,156.075
C06194=1061.641,244.254,408.602,173.006,32.825,156.076
C06195=1061.646,244.502,408.574,173.008,32.829,156.077
C06196=1061.653,244.751,408.546,173.011,32.833,156.078
C06197=1061.659,244.999,408.518,173.013,32.836,156.078
C06198=1061.664,245.247,408.490,173.015,32.840,156.079
C06199=1061.671,245.496,408.462,173.018,32.844,156.080
C06200=1061.677,245.745,408.434,173.020,32.848,156.081
C06201=1061.683,245.993,408.406,173.022,32.852,156.081
C06202=1061.689,246.241,408.378,173.025,32.856,156.082
C06203=1061.696,246.490,408.351,173.027,32.859,156.083
C06204=1061.701,246.738,408.322,173.030,32.864,156.083
C06205=1061.707,246.986,408.294,173.032,32.867,156.084
C06206=1061.713,247.234,408.265,173.034,32.872,156.085
C06207=1061.720,247.483,408.237,173.037,32.875,156.086
C06208=1061.725,247.731,408.210,173.039,32.880,156.086
C06209=1061.731,247.980,408.181,173.041,32.883,156.087
C06210=1061.737,248.228,408.153,173.044,32.888,156.088
C06211=1061.742,248.476,408.125,173.046,32.891,156.089
C06212=1061.748,248.701,408.099,173.048,32.895,156.089
C06213=1061.754,248.925,408.073,173.050,32.898,156.090
C06214=1061.759,249.149,408.048,173.053,32.902,156.091
C06215=1061.765,249.374,408.022,173.055,32.905,156.091
C06216=1061.770,249.598,407.997,173.057,32.909,156.092
C06217=1061.775,249.823,407.972,173.059,32.913,156.093
C06218=1061.781,250.046,407.946,173.061,32.916,156.093
C06219=1061.786,250.271,407.920,173.063,32.919,156.094
C06220=1061.792,250.520,407.892,173.066,32.924,156.095
C06221=1061.798,250.768,407.864,173.068,32.927,156.095
C06222=1061.805,251.016,407.835,173.071,32.932,156.096
C06223=1061.811,251.265,407.807,173.073,32.935,156.097
C06224=1061.817,251.513,407.779,173.075,32.939,156.098
C06225=1061.822,251.761,407.750,173.078,32.943,156.098
C06226=1061.828,252.010,407.722,173.080,32.947,156.099
C06227=1061.835,252.257,407.693,173.083,32.950,156.100
C06228=1061.841,252.506,407.665,173.085,32.955,156.101
C06229=1061.847,252.755,407.637,173.087,32.958,156.101
C06230=1061.853,253.002,407.608,173.090,32.963,156.102
C06231=1061.859,253.251,407.580,173.092,32.966,156.103
C06232=1061.865,253.499,407.550,173.095,32.970,156.103
C06233=1061.872,253.748,407.523,173.097,32.974,156.104
C06234=1061.878,253.996,407.494,173.100,32.978,156.105
C06235=1061.884,254.245,407.465,173.102,32.982,156.106
C06236=1061.890,254.493,407.436,173.105,32.986,156.106
C06237=1061.895,254.741,407.408,173.107,32.989,156.107
C06238=1061.902,254.989,407.379,173.109,32.993,156.108
C06239=1061.908,255.238,407.351,173.112,32.997,156.109
C06240=1061.915,255.485,407.323,173.114,33.001,156.109
C06241=1061.920,255.734,407.294,173.117,33.005,156.110
C06242=1061.927,255.982,407.265,173.119,33.009,156.111
C06243=1061.933,256.231,407.237,173.122,33.013,156.111
C06244=1061.939,256.479,407.208,173.124,33.016,156.112
C06245=1061.945,256.727,407.179,173.127,33.021,156.113
C06246=1061.951,256.976,407.150,173.129,33.024,156.114
C06247=1061.957,257.223,407.122,173.132,33.028,156.114
C06248=1061.964,257.471,407.093,173.134,33.032,156.115
C06249=1061.970,257.720,407.065,173.137,33.036,156.116
C06250=1061.976,257.968,407.036,173.139,33.040,156.117
C06251=1061.982,258.216,407.007,173.142,33.043,156.117
C06252=1061.988,258.465,406.979,173.144,33.047,156.118
C06253=1061.994,258.713,406.950,173.147,33.051,156.119
C06254=1062.001,258.961,406.921,173.149,33.055,156.119
C06255=1062.007,259.209,406.891,173.152,33.059,156.120
C06256=1062.013,259.458,406.863,173.154,33.063,156.121
C06257=1062.019,259.706,406.834,173.157,33.066,156.122
C06258=1062.025,259.954,406.805,173.159,33.070,156.122
C06259=1062.032,260.202,406.777,173.162,33.074,156.123
C06260=1062.038,260.451,406.748,173.164,33.078,156.124
C06261=1062.044,260.699,406.719,173.167,33.082,156.124
C06262=1062.051,260.947,406.690,173.169,33.086,156.125
C06263=1062.058,261.196,406.661,173.172,33.090,156.126
C06264=1062.064,261.444,406.632,173.175,33.093,156.127
C06265=1062.070,261.692,406.603,173.178,33.097,156.127
C06266=1062.076,261.941,406.574,173.180,33.101,156.128
C06267=1062.082,262.189,406.545,173.183,33.105,156.129
C06268=1062.088,262.412,406.519,173.185,33.108,156.129
C06269=1062.094,262.636,406.493,173.187,33.111,156.130
C06270=1062.099,262.860,406.467,173.190,33.115,156.131
C06271=1062.106,263.082,406.440,173.192,33.118,156.131
C06272=1062.111,263.305,406.415,173.194,33.122,156.132
C06273=1062.116,263.529,406.389,173.197,33.126,156.133
C06274=1062.122,263.752,406.362,173.199,33.129,156.133
C06275=1062.127,263.975,406.336,173.201,33.132,156.134
C06276=1062.133,264.224,406.306,173.204,33.136,156.135
C06277=1062.139,264.472,406.277,173.206,33.140,156.136
C06278=1062.145,264.720,406.248,173.209,33.144,156.136
C06279=1062.152,264.968,406.219,173.211,33.148,156.137
C06280=1062.157,265.217,406.190,173.214,33.152,156.138
C06281=1062.164,265.464,406.160,173.216,33.156,156.139
C06282=1062.170,265.712,406.131,173.219,33.160,156.139
C06283=1062.176,265.961,406.101,173.221,33.163,156.140
C06284=1062.182,266.209,406.072,173.224,33.167,156.141
C06285=1062.189,266.458,406.043,173.227,33.171,156.141
C06286=1062.194,266.706,406.013,173.229,33.175,156.142
C06287=1062.200,266.954,405.984,173.232,33.179,156.143
C06288=1062.207,267.202,405.954,173.234,33.183,156.144
C06289=1062.213,267.450,405.925,173.237,33.187,156.144
C06290=1062.219,267.698,405.896,173.239,33.191,156.145
C06291=1062.226,267.947,405.866,173.242,33.195,156.146
C06292=1062.232,268.195,405.837,173.245,33.199,156.147
C06293=1062.238,268.443,405.807,173.247,33.202,156.147
C06294=1062.244,268.691,405.778,173.250,33.206,156.148
C06295=1062.250,268.939,405.748,173.252,33.210,156.149
C06296=1062.256,269.187,405.718,173.255,33.214,156.150
C06297=1062.262,269.435,405.689,173.258,33.218,156.150
C06298=1062.269,269.684,405.659,173.260,33.222,156.151
C06299=1062.275,269.932,405.630,173.263,33.226,156.152
C06300=1062.280,270.180,405.600,173.265,33.229,156.153
C06301=1062.287,270.428,405.570,173.269,33.234,156.153
C06302=1062.292,270.676,405.541,173.272,33.237,156.154
C06303=1062.300,270.925,405.511,173.274,33.242,156.155
C06304=1062.306,271.173,405.481,173.277,33.245,156.156
C06305=1062.311,271.421,405.452,173.279,33.249,156.156
C06306=1062.318,271.669,405.422,173.282,33.253,156.157
C06307=1062.323,271.917,405.392,173.285,33.257,156.158
C06308=1062.331,272.165,405.362,173.287,33.261,156.159
C06309=1062.336,272.414,405.333,173.290,33.265,156.159
C06310=1062.343,272.661,405.303,173.293,33.269,156.160
C06311=1062.348,272.910,405.273,173.295,33.273,156.161
C06312=1062.355,273.158,405.243,173.298,33.277,156.162
C06313=1062.361,273.406,405.213,173.300,33.280,156.162
C06314=1062.367,273.654,405.183,173.303,33.285,156.163
C06315=1062.373,273.902,405.153,173.306,33.288,156.164
C06316=1062.379,274.151,405.123,173.308,33.292,156.165
C06317=1062.385,274.399,405.093,173.311,33.296,156.165
C06318=1062.392,274.646,405.063,173.314,33.300,156.166
C06319=1062.397,274.895,405.034,173.316,33.304,156.167
C06320=1062.404,275.143,405.004,173.319,33.308,156.168
C06321=1062.410,275.391,404.973,173.322,33.312,156.168
C06322=1062.416,275.639,404.944,173.324,33.316,156.169
C06323=1062.423,275.887,404.913,173.327,33.320,156.170
C06324=1062.428,276.112,404.886,173.330,33.323,156.170
C06325=1062.433,276.338,404.859,173.333,33.327,156.171
C06326=1062.439,276.562,404.832,173.335,33.331,156.172
C06327=1062.445,276.788,404.804,173.338,33.334,156.173
C06328=1062.450,277.013,404.776,173.340,33.338,156.173
C06329=1062.455,277.238,404.749,173.342,33.341,156.174
C06330=1062.461,277.463,404.722,173.345,33.345,156.175
C06331=1062.467,277.689,404.695,173.347,33.348,156.175
C06332=1062.473,277.936,404.664,173.350,33.352,156.176
C06333=1062.479,278.184,404.634,173.353,33.356,156.177
C06334=1062.486,278.432,404.604,173.355,33.360,156.178
C06335=1062.492,278.680,404.573,173.358,33.364,156.178
C06336=1062.498,278.929,404.543,173.361,33.368,156.179
C06337=1062.504,279.177,404.513,173.363,33.372,156.180
C06338=1062.511,279.425,404.483,173.366,33.376,156.181
C06339=1062.517,279.673,404.453,173.369,33.380,156.181
C06340=1062.523,279.921,404.422,173.371,33.384,156.182
C06341=1062.529,280.170,404.392,173.374,33.388,156.183
C06342=1062.535,280.417,404.361,173.377,33.392,156.184
C06343=1062.541,280.665,404.331,173.381,33.396,156.184
C06344=1062.548,280.913,404.301,173.383,33.400,156.185
C06345=1062.554,281.161,404.270,173.386,33.404,156.186
C06346=1062.560,281.409,404.240,173.389,33.408,156.187
C06347=1062.566,281.658,404.209,173.391,33.412,156.187
C06348=1062.572,281.905,404.178,173.394,33.416,156.188
C06349=1062.579,282.153,404.147,173.397,33.420,156.189
C06350=1062.584,282.401,404.117,173.400,33.424,156.190
C06351=1062.590,282.649,404.087,173.402,33.427,156.190
C06352=1062.597,282.897,404.056,173.405,33.432,156.191
C06353=1062.602,283.145,404.026,173.408,33.436,156.192
C06354=1062.609,283.394,403.995,173.411,33.440,156.193
C06355=1062.615,283.641,403.964,173.413,33.444,156.194
C06356=1062.621,283.890,403.933,173.416,33.448,156.194
C06357=1062.627,284.137,403.903,173.419,33.452,156.195
C06358=1062.634,284.386,403.872,173.422,33.456,156.196
C06359=1062.639,284.634,403.842,173.425,33.459,156.197
C06360=1062.646,284.882,403.810,173.428,33.464,156.197
C06361=1062.652,285.129,403.780,173.431,33.468,156.198
C06362=1062.658,285.378,403.749,173.434,33.472,156.199
C06363=1062.665,285.625,403.718,173.436,33.476,156.200
C06364=1062.671,285.874,403.688,173.439,33.479,156.201
C06365=1062.677,286.122,403.657,173.442,33.484,156.201
C06366=1062.683,286.369,403.626,173.445,33.488,156.202
C06367=1062.689,286.617,403.595,173.447,33.491,156.203
C06368=1062.696,286.866,403.565,173.450,33.496,156.204
C06369=1062.702,287.113,403.534,173.453,33.499,156.204
C06370=1062.708,287.361,403.503,173.456,33.503,156.205
C06371=1062.715,287.610,403.472,173.460,33.508,156.206
C06372=1062.721,287.857,403.441,173.462,33.511,156.207
C06373=1062.727,288.106,403.410,173.465,33.515,156.208
C06374=1062.733,288.353,403.379,173.468,33.520,156.208
C06375=1062.740,288.601,403.349,173.471,33.523,156.209
C06376=1062.746,288.850,403.317,173.474,33.528,156.210
C06377=1062.752,289.097,403.286,173.476,33.532,156.211
C06378=1062.758,289.345,403.255,173.479,33.535,156.211
C06379=1062.764,289.593,403.224,173.482,33.540,156.212
C06380=1062.770,289.824,403.195,173.485,33.543,156.213
C06381=1062.776,290.055,403.166,173.487,33.547,156.214
C06382=1062.782,290.285,403.137,173.490,33.551,156.214
C06383=1062.788,290.515,403.108,173.492,33.555,156.215
C06384=1062.793,290.746,403.079,173.496,33.558,156.216
C06385=1062.799,290.976,403.050,173.499,33.562,156.217
C06386=1062.805,291.206,403.021,173.501,33.566,156.217
C06387=1062.810,291.437,402.993,173.504,33.570,156.218
C06388=1062.817,291.685,402.961,173.507,33.574,156.219
C06389=1062.823,291.933,402.929,173.510,33.578,156.220
C06390=1062.829,292.180,402.898,173.512,33.582,156.220
C06391=1062.835,292.429,402.867,173.515,33.586,156.221
C06392=1062.841,292.677,402.835,173.518,33.590,156.222
C06393=1062.848,292.924,402.804,173.521,33.594,156.223
C06394=1062.854,293.172,402.773,173.524,33.598,156.224
C06395=1062.860,293.421,402.742,173.528,33.602,156.224
C06396=1062.866,293.668,402.711,173.530,33.606,156.225
C06397=1062.873,293.916,402.679,173.533,33.610,156.226
C06398=1062.879,294.164,402.647,173.536,33.615,156.227
C06399=1062.885,294.412,402.616,173.539,33.618,156.228
C06400=1062.892,294.659,402.585,173.542,33.622,156.228
C06401=1062.897,294.908,402.553,173.545,33.627,156.229
C06402=1062.904,295.156,402.522,173.548,33.631,156.230
C06403=1062.910,295.403,402.491,173.551,33.635,156.231
C06404=1062.916,295.652,402.459,173.553,33.639,156.232
C06405=1062.923,295.900,402.427,173.557,33.643,156.232
C06406=1062.929,296.148,402.395,173.560,33.647,156.233
C06407=1062.935,296.395,402.364,173.563,33.651,156.234
C06408=1062.941,296.643,402.332,173.566,33.655,156.235
C06409=1062.948,296.891,402.301,173.569,33.660,156.236
C06410=1062.954,297.139,402.269,173.572,33.663,156.236
C06411=1062.960,297.386,402.238,173.575,33.667,156.237
C06412=1062.966,297.635,402.206,173.578,33.672,156.238
C06413=1062.972,297.883,402.174,173.580,33.676,156.239
C06414=1062.978,298.131,402.141,173.583,33.680,156.240
C06415=1062.984,298.378,402.110,173.587,33.685,156.241
C06416=1062.990,298.626,402.078,173.590,33.689,156.241
C06417=1062.996,298.874,402.046,173.593,33.693,156.242
C06418=1063.003,299.122,402.014,173.596,33.697,156.243
C06419=1063.008,299.370,401.983,173.599,33.702,156.244
C06420=1063.015,299.617,401.950,173.602,33.706,156.245
C06421=1063.021,299.865,401.918,173.605,33.710,156.246
C06422=1063.027,300.113,401.886,173.608,33.714,156.246
C06423=1063.033,300.361,401.855,173.611,33.718,156.247
C06424=1063.039,300.608,401.822,173.614,33.722,156.248
C06425=1063.045,300.857,401.790,173.617,33.727,156.249
C06426=1063.052,301.104,401.759,173.620,33.731,156.250
C06427=1063.058,301.352,401.726,173.623,33.735,156.251
C06428=1063.063,301.600,401.694,173.626,33.739,156.251
C06429=1063.069,301.848,401.662,173.629,33.743,156.252
C06430=1063.076,302.095,401.629,173.632,33.748,156.253
C06431=1063.082,302.343,401.598,173.635,33.752,156.254
C06432=1063.089,302.591,401.565,173.639,33.756,156.255
C06433=1063.095,302.839,401.533,173.642,33.760,156.256
C06434=1063.101,303.087,401.501,173.645,33.764,156.256
C06435=1063.108,303.335,401.469,173.648,33.768,156.257
C06436=1063.113,303.573,401.438,173.651,33.773,156.258
C06437=1063.119,303.811,401.407,173.653,33.777,156.259
C06438=1063.125,304.049,401.376,173.656,33.781,156.260
C06439=1063.131,304.287,401.345,173.659,33.784,156.260
C06440=1063.137,304.524,401.314,173.663,33.789,156.261
C06441=1063.143,304.763,401.283,173.666,33.793,156.262
C06442=1063.148,305.001,401.252,173.669,33.797,156.263
C06443=1063.155,305.239,401.221,173.672,33.801,156.264
C06444=1063.161,305.487,401.189,173.675,33.805,156.265
C06445=1063.168,305.735,401.157,173.678,33.810,156.265
C06446=1063.174,305.982,401.124,173.681,33.814,156.266
C06447=1063.180,306.231,401.092,173.684,33.818,156.267
C06448=1063.187,306.478,401.059,173.688,33.822,156.268
C06449=1063.193,306.726,401.026,173.691,33.826,156.269
C06450=1063.199,306.974,400.994,173.694,33.830,156.270
C06451=1063.206,307.221,400.962,173.697,33.835,156.270
C06452=1063.212,307.469,400.929,173.700,33.839,156.271
C06453=1063.218,307.717,400.897,173.703,33.843,156.272
C06454=1063.225,307.965,400.865,173.706,33.848,156.273
C06455=1063.231,308.212,400.832,173.710,33.852,156.274
C06456=1063.237,308.460,400.799,173.713,33.856,156.275
C06457=1063.243,308.708,400.767,173.716,33.860,156.275
C06458=1063.249,308.956,400.734,173.719,33.864,156.276
C06459=1063.256,309.203,400.702,173.722,33.869,156.277
C06460=1063.263,309.450,400.670,173.725,33.873,156.278
C06461=1063.270,309.699,400.636,173.728,33.877,156.279
C06462=1063.276,309.946,400.604,173.732,33.882,156.280
C06463=1063.282,310.195,400.572,173.735,33.886,156.281
C06464=1063.288,310.442,400.539,173.738,33.890,156.281
C06465=1063.294,310.690,400.506,173.741,33.894,156.282
C06466=1063.301,310.937,400.473,173.744,33.899,156.283
C06467=1063.308,311.186,400.440,173.748,33.903,156.284
C06468=1063.314,311.433,400.408,173.751,33.907,156.285
C06469=1063.321,311.681,400.375,173.755,33.911,156.286
C06470=1063.327,311.928,400.343,173.758,33.915,156.287
C06471=1063.334,312.176,400.310,173.761,33.920,156.287
C06472=1063.340,312.424,400.277,173.764,33.924,156.288
C06473=1063.347,312.672,400.244,173.767,33.928,156.289
C06474=1063.353,312.919,400.211,173.770,33.933,156.290
C06475=1063.359,313.167,400.179,173.773,33.937,156.291
C06476=1063.366,313.415,400.146,173.777,33.941,156.292
C06477=1063.373,313.663,400.113,173.780,33.946,156.293
C06478=1063.379,313.910,400.080,173.784,33.950,156.293
C06479=1063.385,314.158,400.047,173.787,33.954,156.294
C06480=1063.392,314.406,400.013,173.790,33.959,156.295
C06481=1063.398,314.653,399.980,173.793,33.963,156.296
C06482=1063.403,314.901,399.947,173.797,33.968,156.297
C06483=1063.410,315.149,399.914,173.800,33.972,156.298
C06484=1063.416,315.396,399.880,173.803,33.976,156.299
C06485=1063.422,315.644,399.847,173.806,33.981,156.300
C06486=1063.429,315.892,399.814,173.809,33.985,156.301
C06487=1063.434,316.140,399.781,173.812,33.990,156.302
C06488=1063.441,316.387,399.747,173.816,33.994,156.302
C06489=1063.446,316.635,399.714,173.820,33.999,156.303
C06490=1063.453,316.883,399.681,173.823,34.003,156.304
C06491=1063.459,317.130,399.647,173.826,34.008,156.305
C06492=1063.465,317.370,399.615,173.829,34.012,156.306
C06493=1063.471,317.610,399.582,173.833,34.017,156.307
C06494=1063.478,317.850,399.550,173.836,34.021,156.308
C06495=1063.484,318.090,399.517,173.839,34.025,156.309
C06496=1063.490,318.330,399.486,173.842,34.030,156.310
C06497=1063.495,318.569,399.453,173.845,34.034,156.310
C06498=1063.501,318.810,399.420,173.848,34.038,156.311
C06499=1063.508,319.050,399.388,173.852,34.043,156.312
C06500=1063.513,319.297,399.355,173.855,34.047,156.313
C06501=1063.521,319.545,399.321,173.858,34.051,156.314
C06502=1063.526,319.793,399.287,173.862,34.056,156.315
C06503=1063.533,320.040,399.254,173.865,34.060,156.316
C06504=1063.539,320.288,399.220,173.868,34.065,156.317
C06505=1063.546,320.536,399.187,173.872,34.070,156.318
C06506=1063.552,320.784,399.152,173.875,34.074,156.319
C06507=1063.558,321.031,399.120,173.878,34.078,156.320
C06508=1063.564,321.278,399.086,173.882,34.083,156.320
C06509=1063.571,321.526,399.052,173.885,34.087,156.321
C06510=1063.577,321.774,399.018,173.889,34.092,156.322
C06511=1063.584,322.022,398.985,173.892,34.097,156.323
C06512=1063.590,322.269,398.951,173.895,34.101,156.324
C06513=1063.597,322.517,398.917,173.899,34.106,156.325
C06514=1063.603,322.765,398.883,173.902,34.110,156.326
C06515=1063.609,323.013,398.849,173.906,34.115,156.327
C06516=1063.616,323.260,398.815,173.909,34.119,156.328
C06517=1063.622,323.508,398.781,173.912,34.124,156.329
C06518=1063.629,323.755,398.748,173.916,34.129,156.330
C06519=1063.635,324.003,398.714,173.919,34.133,156.331
C06520=1063.642,324.250,398.680,173.923,34.137,156.332
C06521=1063.648,324.498,398.646,173.926,34.142,156.332
C06522=1063.654,324.745,398.612,173.929,34.147,156.333
C06523=1063.661,324.993,398.578,173.933,34.151,156.334
C06524=1063.667,325.240,398.544,173.936,34.156,156.335
C06525=1063.674,325.489,398.511,173.940,34.160,156.336
C06526=1063.680,325.736,398.477,173.943,34.165,156.337
C06527=1063.686,325.984,398.443,173.947,34.170,156.338
C06528=1063.693,326.232,398.409,173.950,34.174,156.339
C06529=1063.699,326.479,398.375,173.953,34.178,156.340
C06530=1063.706,326.726,398.341,173.958,34.183,156.341
C06531=1063.713,326.974,398.306,173.961,34.188,156.342
C06532=1063.719,327.222,398.272,173.964,34.193,156.343
C06533=1063.726,327.469,398.239,173.967,34.197,156.344
C06534=1063.733,327.717,398.203,173.972,34.201,156.345
C06535=1063.739,327.964,398.170,173.975,34.206,156.346
C06536=1063.746,328.212,398.136,173.978,34.211,156.347
C06537=1063.752,328.460,398.101,173.981,34.215,156.348
C06538=1063.759,328.707,398.068,173.985,34.220,156.349
C06539=1063.765,328.955,398.033,173.989,34.225,156.349
C06540=1063.772,329.203,397.999,173.992,34.229,156.350
C06541=1063.779,329.449,397.965,173.996,34.234,156.351
C06542=1063.785,329.697,397.930,173.999,34.239,156.352
C06543=1063.792,329.945,397.896,174.003,34.243,156.353
C06544=1063.799,330.193,397.862,174.007,34.248,156.354
C06545=1063.805,330.441,397.828,174.010,34.252,156.355
C06546=1063.811,330.687,397.793,174.013,34.257,156.356
C06547=1063.818,330.935,397.758,174.017,34.262,156.357
C06548=1063.824,331.173,397.725,174.021,34.266,156.358
C06549=1063.830,331.409,397.692,174.024,34.271,156.359
C06550=1063.836,331.647,397.659,174.027,34.276,156.360
C06551=1063.842,331.884,397.626,174.030,34.280,156.361
C06552=1063.849,332.121,397.593,174.035,34.285,156.362
C06553=1063.855,332.357,397.560,174.038,34.289,156.363
C06554=1063.861,332.595,397.526,174.041,34.294,156.364
C06555=1063.867,332.831,397.493,174.044,34.298,156.365
C06556=1063.874,333.079,397.458,174.048,34.303,156.366
C06557=1063.880,333.327,397.424,174.052,34.308,156.367
C06558=1063.887,333.574,397.389,174.055,34.313,156.368
C06559=1063.893,333.821,397.355,174.059,34.318,156.369
C06560=1063.900,334.069,397.319,174.063,34.322,156.370
C06561=1063.906,334.317,397.285,174.066,34.328,156.371
C06562=1063.913,334.564,397.250,174.070,34.332,156.372
C06563=1063.920,334.811,397.215,174.073,34.337,156.373
C06564=1063.926,335.059,397.180,174.077,34.342,156.374
C06565=1063.932,335.306,397.146,174.081,34.347,156.375
C06566=1063.939,335.553,397.110,174.084,34.351,156.376
C06567=1063.945,335.802,397.075,174.088,34.356,156.377
C06568=1063.951,336.049,397.040,174.092,34.361,156.378
C06569=1063.958,336.296,397.005,174.095,34.366,156.379
C06570=1063.965,336.544,396.971,174.099,34.371,156.380
C06571=1063.971,336.792,396.936,174.102,34.376,156.381
C06572=1063.978,337.039,396.900,174.107,34.381,156.382
C06573=1063.985,337.286,396.865,174.110,34.386,156.383
C06574=1063.991,337.533,396.831,174.113,34.390,156.384
C06575=1063.997,337.781,396.795,174.117,34.396,156.385
C06576=1064.004,338.029,396.760,174.121,34.400,156.386
C06577=1064.010,338.276,396.725,174.125,34.406,156.387
C06578=1064.016,338.524,396.690,174.128,34.410,156.388
C06579=1064.023,338.771,396.654,174.132,34.415,156.389
C06580=1064.030,339.019,396.619,174.136,34.421,156.390
C06581=1064.036,339.266,396.584,174.139,34.425,156.391
C06582=1064.043,339.514,396.548,174.143,34.430,156.392
C06583=1064.050,339.761,396.513,174.147,34.435,156.393
C06584=1064.056,340.008,396.478,174.151,34.440,156.394
C06585=1064.062,340.256,396.442,174.154,34.445,156.396
C06586=1064.069,340.503,396.407,174.159,34.450,156.397
C06587=1064.076,340.751,396.372,174.162,34.455,156.398
C06588=1064.082,340.998,396.336,174.166,34.461,156.399
C06589=1064.089,341.245,396.301,174.169,34.465,156.400
C06590=1064.096,341.492,396.265,174.173,34.470,156.401
C06591=1064.102,341.740,396.230,174.177,34.476,156.402
C06592=1064.109,341.988,396.195,174.180,34.480,156.403
C06593=1064.115,342.235,396.159,174.185,34.485,156.404
C06594=1064.122,342.482,396.123,174.188,34.491,156.405
C06595=1064.128,342.729,396.088,174.192,34.495,156.406
C06596=1064.134,342.977,396.052,174.195,34.500,156.407
C06597=1064.141,343.224,396.017,174.200,34.506,156.408
C06598=1064.148,343.471,395.981,174.203,34.511,156.409
C06599=1064.155,343.719,395.945,174.207,34.516,156.410
C06600=1064.162,343.967,395.910,174.211,34.521,156.411
C06601=1064.168,344.214,395.873,174.215,34.526,156.413
C06602=1064.175,344.461,395.838,174.218,34.531,156.414
C06603=1064.181,344.709,395.803,174.223,34.536,156.415
C06604=1064.187,344.944,395.769,174.226,34.541,156.416
C06605=1064.193,345.178,395.735,174.230,34.546,156.417
C06606=1064.200,345.413,395.701,174.234,34.551,156.418
C06607=1064.206,345.648,395.666,174.237,34.556,156.419
C06608=1064.212,345.882,395.632,174.241,34.561,156.420
C06609=1064.219,346.116,395.598,174.244,34.566,156.421
C06610=1064.225,346.351,395.564,174.248,34.571,156.422
C06611=1064.231,346.586,395.530,174.252,34.576,156.423
C06612=1064.237,346.834,395.494,174.255,34.581,156.424
C06613=1064.244,347.080,395.458,174.260,34.586,156.425
C06614=1064.250,347.327,395.422,174.263,34.592,156.427
C06615=1064.258,347.575,395.386,174.267,34.597,156.428
C06616=1064.264,347.822,395.350,174.272,34.602,156.429
C06617=1064.270,348.069,395.313,174.275,34.607,156.430
C06618=1064.276,348.317,395.277,174.279,34.612,156.431
C06619=1064.284,348.565,395.241,174.283,34.618,156.432
C06620=1064.290,348.812,395.205,174.287,34.623,156.433
C06621=1064.297,349.059,395.168,174.291,34.628,156.434
C06622=1064.304,349.306,395.133,174.295,34.634,156.436
C06623=1064.311,349.554,395.096,174.299,34.639,156.437
C06624=1064.317,349.801,395.060,174.302,34.644,156.438
C06625=1064.323,350.048,395.024,174.307,34.650,156.439
C06626=1064.330,350.295,394.988,174.311,34.655,156.440
C06627=1064.337,350.542,394.951,174.315,34.661,156.441
C06628=1064.343,350.790,394.915,174.319,34.666,156.442
C06629=1064.350,351.037,394.879,174.322,34.671,156.444
C06630=1064.357,351.285,394.842,174.327,34.676,156.445
C06631=1064.364,351.532,394.806,174.331,34.682,156.446
C06632=1064.371,351.779,394.769,174.334,34.687,156.447
C06633=1064.377,352.026,394.733,174.339,34.693,156.448
C06634=1064.383,352.274,394.696,174.343,34.698,156.449
C06635=1064.391,352.521,394.660,174.346,34.704,156.451
C06636=1064.397,352.768,394.624,174.351,34.709,156.452
C06637=1064.404,353.014,394.586,174.355,34.714,156.453
C06638=1064.411,353.262,394.550,174.359,34.720,156.454
C06639=1064.417,353.509,394.513,174.363,34.725,156.455
C06640=1064.423,353.756,394.477,174.367,34.731,156.456
C06641=1064.430,354.004,394.440,174.371,34.736,156.458
C06642=1064.437,354.251,394.404,174.375,34.742,156.459
C06643=1064.444,354.498,394.366,174.379,34.747,156.460
C06644=1064.450,354.745,394.330,174.383,34.753,156.461
C06645=1064.457,354.993,394.293,174.387,34.758,156.462
C06646=1064.464,355.240,394.256,174.392,34.764,156.464
C06647=1064.470,355.487,394.219,174.395,34.769,156.465
C06648=1064.477,355.734,394.182,174.399,34.775,156.466
C06649=1064.484,355.981,394.145,174.404,34.780,156.467
C06650=1064.491,356.229,394.108,174.407,34.786,156.468
C06651=1064.497,356.476,394.072,174.412,34.792,156.470
C06652=1064.504,356.723,394.034,174.416,34.797,156.471
C06653=1064.511,356.970,393.998,174.420,34.803,156.472
C06654=1064.518,357.217,393.960,174.424,34.808,156.473
C06655=1064.525,357.465,393.924,174.428,34.814,156.475
C06656=1064.531,357.711,393.886,174.433,34.820,156.476
C06657=1064.538,357.959,393.850,174.437,34.825,156.477
C06658=1064.545,358.205,393.812,174.440,34.831,156.478
C06659=1064.552,358.453,393.776,174.445,34.837,156.479
C06660=1064.558,358.689,393.740,174.449,34.842,156.481
C06661=1064.565,358.927,393.704,174.453,34.847,156.482
C06662=1064.571,359.163,393.668,174.457,34.853,156.483
C06663=1064.578,359.400,393.633,174.461,34.858,156.484
C06664=1064.584,359.636,393.597,174.465,34.864,156.485
C06665=1064.591,359.873,393.562,174.469,34.869,156.487
C06666=1064.597,360.110,393.525,174.473,34.875,156.488
C06667=1064.603,360.346,393.490,174.477,34.880,156.489
C06668=1064.610,360.594,393.452,174.482,34.886,156.490
C06669=1064.618,360.841,393.415,174.486,34.892,156.492
C06670=1064.624,361.087,393.378,174.489,34.897,156.493
C06671=1064.631,361.335,393.340,174.494,34.903,156.494
C06672=1064.638,361.582,393.303,174.498,34.909,156.495
C06673=1064.644,361.829,393.266,174.503,34.915,156.497
C06674=1064.652,362.076,393.228,174.507,34.921,156.498
C06675=1064.658,362.323,393.190,174.511,34.926,156.499
C06676=1064.665,362.570,393.153,174.515,34.933,156.501
C06677=1064.672,362.817,393.115,174.520,34.938,156.502
C06678=1064.678,363.064,393.077,174.524,34.944,156.503
C06679=1064.686,363.312,393.040,174.529,34.950,156.504
C06680=1064.692,363.558,393.003,174.533,34.956,156.506
C06681=1064.699,363.805,392.964,174.536,34.961,156.507
C06682=1064.706,364.053,392.927,174.541,34.968,156.508
C06683=1064.713,364.300,392.889,174.545,34.973,156.510
C06684=1064.719,364.546,392.852,174.550,34.980,156.511
C06685=1064.727,364.793,392.813,174.554,34.985,156.512
C06686=1064.733,365.040,392.775,174.559,34.991,156.514
C06687=1064.741,365.288,392.738,174.563,34.998,156.515
C06688=1064.746,365.534,392.700,174.567,35.003,156.516
C06689=1064.754,365.781,392.662,174.571,35.010,156.518
C06690=1064.760,366.028,392.624,174.576,35.016,156.519
C06691=1064.767,366.276,392.585,174.580,35.021,156.520
C06692=1064.774,366.523,392.548,174.585,35.028,156.522
C06693=1064.780,366.769,392.509,174.589,35.034,156.523
C06694=1064.788,367.016,392.472,174.594,35.039,156.524
C06695=1064.794,367.263,392.433,174.598,35.046,156.526
C06696=1064.802,367.510,392.396,174.603,35.052,156.527
C06697=1064.808,367.757,392.357,174.606,35.058,156.528
C06698=1064.815,368.004,392.319,174.611,35.064,156.530
C06699=1064.822,368.251,392.281,174.615,35.070,156.531
C06700=1064.829,368.498,392.242,174.620,35.076,156.532
C06701=1064.836,368.745,392.205,174.624,35.082,156.534
C06702=1064.843,368.991,392.166,174.629,35.088,156.535
C06703=1064.849,369.238,392.127,174.633,35.095,156.537
C06704=1064.857,369.485,392.090,174.638,35.101,156.538
C06705=1064.863,369.732,392.051,174.642,35.107,156.539
C06706=1064.871,369.979,392.014,174.647,35.113,156.541
C06707=1064.877,370.226,391.975,174.652,35.119,156.542
C06708=1064.884,370.473,391.936,174.656,35.126,156.543
C06709=1064.892,370.720,391.898,174.661,35.132,156.545
C06710=1064.898,370.967,391.859,174.665,35.138,156.546
C06711=1064.905,371.214,391.821,174.670,35.145,156.548
C06712=1064.913,371.460,391.782,174.674,35.151,156.549
C06713=1064.920,371.707,391.744,174.679,35.157,156.551
C06714=1064.927,371.954,391.706,174.683,35.163,156.552
C06715=1064.934,372.202,391.667,174.688,35.169,156.553
C06716=1064.944,372.551,391.613,174.695,35.178,156.555
C06717=1064.954,372.899,391.557,174.700,35.187,156.557
C06718=1064.964,373.248,391.503,174.707,35.196,156.559
C06719=1064.973,373.596,391.447,174.714,35.206,156.562
C06720=1064.980,373.843,391.409,174.719,35.212,156.563
C06721=1064.987,374.089,391.370,174.723,35.219,156.564
C06722=1064.994,374.336,391.332,174.728,35.225,156.566
C06723=1065.001,374.583,391.293,174.732,35.232,156.567
C06724=1065.008,374.831,391.254,174.737,35.238,156.569
C06725=1065.015,375.077,391.215,174.742,35.244,156.570
C06726=1065.022,375.324,391.176,174.746,35.251,156.572
C06727=1065.029,375.570,391.136,174.751,35.257,156.573
C06728=1065.036,375.817,391.097,174.755,35.264,156.575
C06729=1065.043,376.064,391.059,174.760,35.271,156.576
C06730=1065.050,376.311,391.020,174.765,35.277,156.578
C06731=1065.057,376.558,390.980,174.769,35.284,156.579
C06732=1065.068,376.947,390.919,174.777,35.294,156.582
C06733=1065.079,377.336,390.856,174.784,35.305,156.584
C06734=1065.090,377.725,390.795,174.792,35.315,156.586
C06735=1065.102,378.113,390.733,174.799,35.325,156.589
C06736=1065.109,378.361,390.694,174.804,35.332,156.590
C06737=1065.116,378.607,390.655,174.808,35.339,156.592
C06738=1065.123,378.854,390.616,174.814,35.345,156.593
C06739=1065.131,379.101,390.576,174.819,35.352,156.595
C06740=1065.138,379.347,390.536,174.823,35.359,156.596
C06741=1065.145,379.594,390.497,174.828,35.365,156.598
C06742=1065.152,379.841,390.458,174.833,35.372,156.599
C06743=1065.158,380.088,390.418,174.837,35.379,156.601
C06744=1065.166,380.334,390.379,174.843,35.386,156.603
C06745=1065.173,380.581,390.339,174.848,35.393,156.604
C06746=1065.180,380.828,390.300,174.852,35.399,156.606
C06747=1065.188,381.075,390.260,174.857,35.406,156.607
C06748=1065.195,381.321,390.220,174.862,35.413,156.609
C06749=1065.202,381.567,390.181,174.867,35.420,156.610
C06750=1065.209,381.814,390.140,174.872,35.427,156.612
C06751=1065.216,382.060,390.101,174.877,35.434,156.614
C06752=1065.224,382.307,390.061,174.882,35.441,156.615
C06753=1065.230,382.554,390.021,174.886,35.448,156.617
C06754=1065.237,382.801,389.982,174.892,35.455,156.618
C06755=1065.245,383.048,389.942,174.897,35.462,156.620
C06756=1065.251,383.294,389.902,174.901,35.469,156.622
C06757=1065.259,383.541,389.862,174.906,35.476,156.623
C06758=1065.266,383.787,389.822,174.912,35.483,156.625
C06759=1065.273,384.034,389.781,174.916,35.490,156.626
C06760=1065.280,384.280,389.741,174.921,35.497,156.628
C06761=1065.287,384.527,389.701,174.926,35.504,156.630
C06762=1065.294,384.773,389.661,174.932,35.511,156.631
C06763=1065.302,385.020,389.621,174.936,35.519,156.633
C06764=1065.309,385.267,389.581,174.941,35.525,156.635
C06765=1065.317,385.513,389.541,174.946,35.532,156.636
C06766=1065.323,385.760,389.501,174.952,35.540,156.638
C06767=1065.331,386.006,389.461,174.956,35.547,156.640
C06768=1065.339,386.281,389.416,174.962,35.555,156.642
C06769=1065.347,386.555,389.371,174.968,35.563,156.643
C06770=1065.355,386.830,389.326,174.973,35.571,156.645
C06771=1065.363,387.105,389.282,174.979,35.579,156.647
C06772=1065.371,387.351,389.240,174.985,35.586,156.649
C06773=1065.378,387.598,389.201,174.989,35.594,156.651
C06774=1065.385,387.844,389.160,174.994,35.601,156.652
C06775=1065.393,388.091,389.120,175.000,35.608,156.654
C06776=1065.400,388.337,389.079,175.005,35.615,156.656
C06777=1065.407,388.584,389.039,175.010,35.623,156.657
C06778=1065.415,388.830,388.998,175.015,35.630,156.659
C06779=1065.422,389.077,388.958,175.020,35.637,156.661
C06780=1065.430,389.323,388.918,175.026,35.645,156.663
C06781=1065.437,389.570,388.876,175.031,35.652,156.664
C06782=1065.445,389.816,388.836,175.036,35.660,156.666
C06783=1065.452,390.063,388.795,175.041,35.667,156.668
C06784=1065.460,390.309,388.754,175.046,35.674,156.669
C06785=1065.467,390.555,388.714,175.052,35.682,156.671
C06786=1065.474,390.802,388.673,175.057,35.689,156.673
C06787=1065.482,391.049,388.632,175.063,35.697,156.675
C06788=1065.489,391.295,388.591,175.067,35.704,156.676
C06789=1065.496,391.542,388.550,175.072,35.712,156.678
C06790=1065.504,391.787,388.510,175.078,35.719,156.680
C06791=1065.511,392.034,388.469,175.083,35.727,156.682
C06792=1065.518,392.281,388.427,175.089,35.735,156.684
C06793=1065.526,392.527,388.386,175.094,35.742,156.685
C06794=1065.534,392.774,388.345,175.100,35.750,156.687
C06795=1065.541,393.020,388.304,175.105,35.758,156.689
C06796=1065.548,393.267,388.263,175.110,35.766,156.691
C06797=1065.556,393.513,388.222,175.115,35.773,156.693
C06798=1065.564,393.760,388.181,175.121,35.781,156.695
C06799=1065.571,394.006,388.139,175.126,35.788,156.696
C06800=1065.578,394.251,388.098,175.132,35.796,156.698
C06801=1065.585,394.498,388.057,175.137,35.804,156.700
C06802=1065.592,394.745,388.016,175.143,35.812,156.702
C06803=1065.600,394.991,387.974,175.148,35.820,156.704
C06804=1065.607,395.237,387.933,175.154,35.828,156.706
C06805=1065.615,395.484,387.891,175.159,35.835,156.708
C06806=1065.622,395.730,387.849,175.165,35.844,156.709
C06807=1065.630,395.977,387.808,175.170,35.851,156.711
C06808=1065.638,396.223,387.767,175.175,35.859,156.713
C06809=1065.646,396.469,387.725,175.181,35.867,156.715
C06810=1065.653,396.716,387.684,175.186,35.875,156.717
C06811=1065.661,396.962,387.642,175.192,35.883,156.719
C06812=1065.668,397.209,387.601,175.197,35.891,156.721
C06813=1065.675,397.454,387.559,175.203,35.899,156.723
C06814=1065.683,397.701,387.518,175.208,35.907,156.725
C06815=1065.691,397.948,387.475,175.214,35.915,156.727
C06816=1065.699,398.194,387.433,175.220,35.923,156.728
C06817=1065.705,398.441,387.392,175.225,35.931,156.730
C06818=1065.713,398.687,387.350,175.231,35.940,156.732
C06819=1065.720,398.933,387.308,175.237,35.948,156.734
C06820=1065.728,399.179,387.265,175.242,35.956,156.736
C06821=1065.736,399.426,387.224,175.248,35.964,156.738
C06822=1065.743,399.672,387.182,175.253,35.973,156.740
C06823=1065.751,399.918,387.140,175.259,35.981,156.742
C06824=1065.760,400.209,387.090,175.267,35.991,156.745
C06825=1065.769,400.500,387.040,175.273,36.000,156.747
C06826=1065.778,400.792,386.991,175.280,36.010,156.749
C06827=1065.786,401.082,386.941,175.286,36.020,156.752
C06828=1065.795,401.329,386.899,175.292,36.029,156.754
C06829=1065.802,401.575,386.857,175.298,36.037,156.756
C06830=1065.810,401.821,386.815,175.303,36.045,156.758
C06831=1065.817,402.068,386.772,175.309,36.053,156.760
C06832=1065.825,402.314,386.730,175.316,36.062,156.762
C06833=1065.833,402.560,386.687,175.322,36.070,156.764
C06834=1065.841,402.806,386.645,175.327,36.079,156.766
C06835=1065.848,403.053,386.602,175.333,36.088,156.768
C06836=1065.856,403.299,386.560,175.339,36.096,156.770
C06837=1065.864,403.545,386.517,175.345,36.104,156.772
C06838=1065.871,403.791,386.475,175.350,36.113,156.774
C06839=1065.879,404.038,386.432,175.356,36.122,156.776
C06840=1065.887,404.283,386.390,175.362,36.130,156.778
C06841=1065.895,404.530,386.347,175.369,36.139,156.781
C06842=1065.903,404.775,386.304,175.375,36.147,156.783
C06843=1065.910,405.022,386.261,175.381,36.157,156.785
C06844=1065.918,405.268,386.219,175.386,36.165,156.787
C06845=1065.926,405.515,386.176,175.392,36.174,156.789
C06846=1065.933,405.760,386.133,175.398,36.183,156.791
C06847=1065.941,406.007,386.090,175.405,36.192,156.793
C06848=1065.949,406.253,386.047,175.411,36.200,156.796
C06849=1065.956,406.499,386.004,175.417,36.209,156.798
C06850=1065.965,406.745,385.961,175.423,36.218,156.800
C06851=1065.972,406.991,385.918,175.428,36.227,156.802
C06852=1065.980,407.237,385.874,175.435,36.236,156.804
C06853=1065.988,407.483,385.831,175.441,36.245,156.807
C06854=1065.995,407.730,385.789,175.447,36.254,156.809
C06855=1066.003,407.976,385.745,175.453,36.263,156.811
C06856=1066.011,408.222,385.702,175.460,36.272,156.813
C06857=1066.019,408.469,385.659,175.466,36.281,156.815
C06858=1066.026,408.714,385.615,175.472,36.290,156.818
C06859=1066.035,408.960,385.572,175.478,36.299,156.820
C06860=1066.043,409.207,385.529,175.485,36.308,156.822
C06861=1066.050,409.453,385.485,175.491,36.317,156.824
C06862=1066.058,409.698,385.442,175.497,36.327,156.827
C06863=1066.066,409.945,385.399,175.504,36.336,156.829
C06864=1066.074,410.191,385.355,175.510,36.345,156.831
C06865=1066.082,410.437,385.311,175.516,36.354,156.834
C06866=1066.090,410.683,385.268,175.522,36.364,156.836
C06867=1066.098,410.929,385.224,175.529,36.373,156.838
C06868=1066.106,411.176,385.181,175.535,36.382,156.840
C06869=1066.115,411.421,385.137,175.541,36.392,156.843
C06870=1066.122,411.667,385.094,175.548,36.401,156.845
C06871=1066.130,411.913,385.050,175.554,36.411,156.847
C06872=1066.138,412.159,385.006,175.560,36.420,156.850
C06873=1066.146,412.405,384.963,175.568,36.429,156.852
C06874=1066.154,412.651,384.918,175.574,36.439,156.854
C06875=1066.162,412.897,384.875,175.581,36.448,156.857
C06876=1066.170,413.143,384.830,175.587,36.458,156.859
C06877=1066.178,413.390,384.786,175.593,36.467,156.862
C06878=1066.187,413.635,384.743,175.600,36.477,156.864
C06879=1066.195,413.882,384.699,175.607,36.486,156.866
C06880=1066.204,414.176,384.646,175.615,36.498,156.869
C06881=1066.215,414.472,384.593,175.623,36.510,156.872
C06882=1066.224,414.767,384.540,175.630,36.522,156.875
C06883=1066.234,415.063,384.487,175.639,36.533,156.878
C06884=1066.241,415.309,384.442,175.646,36.543,156.880
C06885=1066.249,415.555,384.398,175.652,36.553,156.883
C06886=1066.258,415.801,384.354,175.659,36.562,156.885
C06887=1066.266,416.046,384.309,175.666,36.573,156.888
C06888=1066.274,416.293,384.265,175.673,36.582,156.890
C06889=1066.282,416.539,384.220,175.679,36.592,156.893
C06890=1066.290,416.784,384.176,175.686,36.602,156.895
C06891=1066.299,417.030,384.132,175.693,36.612,156.898
C06892=1066.307,417.276,384.086,175.700,36.622,156.900
C06893=1066.316,417.522,384.042,175.706,36.632,156.903
C06894=1066.323,417.768,383.997,175.714,36.642,156.906
C06895=1066.331,418.013,383.953,175.720,36.652,156.908
C06896=1066.340,418.260,383.908,175.728,36.663,156.911
C06897=1066.348,418.505,383.863,175.735,36.673,156.913
C06898=1066.356,418.751,383.819,175.741,36.683,156.916
C06899=1066.365,418.997,383.774,175.749,36.693,156.918
C06900=1066.373,419.242,383.729,175.755,36.703,156.921
C06901=1066.381,419.489,383.684,175.763,36.714,156.924
C06902=1066.389,419.734,383.639,175.770,36.724,156.926
C06903=1066.398,419.980,383.594,175.776,36.734,156.929
C06904=1066.406,420.226,383.549,175.784,36.744,156.931
C06905=1066.415,420.472,383.504,175.791,36.755,156.934
C06906=1066.423,420.718,383.458,175.798,36.765,156.937
C06907=1066.432,420.964,383.413,175.805,36.776,156.940
C06908=1066.440,421.209,383.369,175.813,36.786,156.942
C06909=1066.447,421.455,383.323,175.819,36.797,156.945
C06910=1066.456,421.701,383.278,175.827,36.807,156.948
C06911=1066.464,421.946,383.232,175.835,36.818,156.950
C06912=1066.473,422.192,383.187,175.842,36.829,156.953
C06913=1066.482,422.438,383.141,175.849,36.839,156.956
C06914=1066.490,422.683,383.095,175.856,36.850,156.959
C06915=1066.499,422.929,383.050,175.864,36.861,156.961
C06916=1066.506,423.174,383.004,175.871,36.871,156.964
C06917=1066.515,423.420,382.959,175.879,36.882,156.967
C06918=1066.524,423.666,382.913,175.886,36.893,156.970
C06919=1066.532,423.911,382.868,175.893,36.904,156.972
C06920=1066.540,424.158,382.822,175.901,36.915,156.975
C06921=1066.549,424.403,382.776,175.909,36.926,156.978
C06922=1066.557,424.648,382.730,175.916,36.936,156.981
C06923=1066.566,424.894,382.685,175.924,36.947,156.984
C06924=1066.574,425.140,382.639,175.931,36.958,156.986
C06925=1066.584,425.385,382.593,175.939,36.969,156.989
C06926=1066.591,425.631,382.547,175.946,36.980,156.992
C06927=1066.600,425.876,382.501,175.954,36.991,156.995
C06928=1066.609,426.122,382.455,175.962,37.003,156.998
C06929=1066.618,426.367,382.409,175.970,37.014,157.001
C06930=1066.626,426.613,382.363,175.977,37.025,157.004
C06931=1066.636,426.859,382.316,175.985,37.036,157.007
C06932=1066.644,427.105,382.270,175.993,37.047,157.010
C06933=1066.652,427.350,382.224,176.001,37.059,157.013
C06934=1066.661,427.595,382.178,176.009,37.070,157.016
C06935=1066.670,427.840,382.131,176.017,37.081,157.018
C06936=1066.680,428.156,382.072,176.026,37.096,157.022
C06937=1066.692,428.471,382.013,176.037,37.111,157.026
C06938=1066.703,428.786,381.952,176.047,37.126,157.030
C06939=1066.714,429.101,381.893,176.057,37.141,157.034
C06940=1066.722,429.346,381.846,176.065,37.152,157.037
C06941=1066.732,429.592,381.799,176.073,37.164,157.040
C06942=1066.741,429.837,381.752,176.082,37.176,157.043
C06943=1066.750,430.083,381.706,176.090,37.187,157.046
C06944=1066.758,430.328,381.659,176.098,37.199,157.049
C06945=1066.767,430.574,381.612,176.106,37.210,157.052
C06946=1066.776,430.818,381.565,176.114,37.222,157.055
C06947=1066.785,431.064,381.519,176.122,37.234,157.059
C06948=1066.793,431.309,381.472,176.130,37.246,157.062
C06949=1066.803,431.555,381.424,176.139,37.258,157.065
C06950=1066.811,431.800,381.377,176.147,37.270,157.068
C06951=1066.820,432.045,381.330,176.155,37.282,157.071
C06952=1066.829,432.291,381.283,176.163,37.294,157.074
C06953=1066.838,432.536,381.236,176.172,37.306,157.078
C06954=1066.847,432.781,381.188,176.180,37.318,157.081
C06955=1066.856,433.027,381.141,176.189,37.330,157.084
C06956=1066.864,433.272,381.093,176.197,37.343,157.087
C06957=1066.873,433.517,381.046,176.206,37.355,157.091
C06958=1066.882,433.762,380.998,176.214,37.367,157.094
C06959=1066.891,434.008,380.951,176.222,37.379,157.097
C06960=1066.899,434.253,380.904,176.232,37.392,157.100
C06961=1066.909,434.498,380.856,176.240,37.404,157.104
C06962=1066.918,434.743,380.808,176.249,37.416,157.107
C06963=1066.927,434.989,380.761,176.257,37.429,157.110
C06964=1066.936,435.234,380.713,176.266,37.442,157.114
C06965=1066.946,435.479,380.665,176.275,37.454,157.117
C06966=1066.955,435.724,380.617,176.283,37.466,157.121
C06967=1066.963,435.970,380.569,176.293,37.479,157.124
C06968=1066.972,436.214,380.521,176.301,37.492,157.127
C06969=1066.982,436.460,380.474,176.310,37.505,157.131
C06970=1066.991,436.704,380.425,176.319,37.517,157.134
C06971=1067.000,436.950,380.378,176.328,37.530,157.138
C06972=1067.010,437.195,380.329,176.337,37.543,157.141
C06973=1067.019,437.440,380.282,176.346,37.555,157.145
C06974=1067.028,437.685,380.233,176.355,37.568,157.148
C06975=1067.037,437.931,380.185,176.364,37.582,157.152
C06976=1067.046,438.175,380.137,176.373,37.594,157.155
C06977=1067.056,438.421,380.089,176.382,37.607,157.159
C06978=1067.065,438.666,380.040,176.392,37.621,157.162
C06979=1067.075,438.911,379.991,176.401,37.633,157.166
C06980=1067.084,439.155,379.943,176.410,37.647,157.169
C06981=1067.093,439.400,379.894,176.419,37.660,157.173
C06982=1067.102,439.646,379.846,176.429,37.673,157.177
C06983=1067.111,439.891,379.797,176.437,37.687,157.180
C06984=1067.121,440.136,379.749,176.447,37.700,157.184
C06985=1067.130,440.380,379.700,176.457,37.713,157.187
C06986=1067.140,440.625,379.650,176.466,37.726,157.191
C06987=1067.149,440.870,379.602,176.476,37.740,157.195
C06988=1067.158,441.115,379.553,176.485,37.753,157.199
C06989=1067.168,441.360,379.504,176.494,37.767,157.202
C06990=1067.177,441.606,379.455,176.504,37.781,157.206
C06991=1067.187,441.850,379.406,176.514,37.794,157.210
C06992=1067.198,442.128,379.350,176.525,37.810,157.214
C06993=1067.208,442.407,379.294,176.536,37.826,157.218
C06994=1067.219,442.685,379.238,176.547,37.841,157.223
C06995=1067.230,442.963,379.182,176.558,37.857,157.227
C06996=1067.240,443.208,379.133,176.568,37.871,157.231
C06997=1067.249,443.453,379.083,176.578,37.885,157.235
C06998=1067.259,443.697,379.034,176.587,37.899,157.239
C06999=1067.269,443.942,378.984,176.597,37.913,157.242
C07000=1067.278,444.188,378.935,176.608,37.927,157.246
C07001=1067.288,444.432,378.885,176.618,37.941,157.250
C07002=1067.298,444.677,378.836,176.628,37.955,157.254
C07003=1067.307,444.921,378.786,176.638,37.969,157.258
C07004=1067.317,445.167,378.736,176.648,37.984,157.262
C07005=1067.326,445.411,378.686,176.658,37.998,157.266
C07006=1067.336,445.656,378.637,176.668,38.012,157.270
C07007=1067.346,445.900,378.586,176.679,38.027,157.274
C07008=1067.356,446.145,378.536,176.689,38.041,157.278
C07009=1067.365,446.390,378.486,176.700,38.056,157.282
C07010=1067.376,446.634,378.436,176.710,38.070,157.287
C07011=1067.385,446.879,378.386,176.721,38.085,157.291
C07012=1067.395,447.124,378.336,176.731,38.100,157.295
C07013=1067.405,447.368,378.285,176.741,38.114,157.299
C07014=1067.415,447.613,378.236,176.752,38.129,157.303
C07015=1067.425,447.857,378.185,176.763,38.144,157.307
C07016=1067.436,448.101,378.135,176.774,38.159,157.311
C07017=1067.447,448.344,378.086,176.784,38.173,157.315
C07018=1067.460,448.589,378.038,176.795,38.187,157.319
C07019=1067.474,448.834,377.989,176.805,38.200,157.323
C07020=1067.488,449.079,377.942,176.815,38.213,157.327
C07021=1067.504,449.324,377.896,176.825,38.226,157.331
C07022=1067.521,449.569,377.850,176.835,38.239,157.334
C07023=1067.539,449.814,377.805,176.845,38.251,157.338
C07024=1067.195,449.818,377.545,176.834,38.382,157.373
C07025=1067.177,449.572,377.589,176.825,38.370,157.369
C07026=1067.161,449.327,377.635,176.815,38.358,157.366
C07027=1067.145,449.082,377.682,176.805,38.345,157.362
C07028=1067.129,448.837,377.730,176.794,38.332,157.359
C07029=1067.115,448.592,377.777,176.784,38.318,157.355
C07030=1067.103,448.348,377.826,176.772,38.304,157.351
C07031=1067.092,448.103,377.875,176.762,38.290,157.347
C07032=1067.080,447.861,377.925,176.750,38.276,157.342
C07033=1067.071,447.616,377.975,176.740,38.260,157.338
C07034=1067.061,447.371,378.025,176.729,38.246,157.334
C07035=1067.050,447.127,378.075,176.719,38.231,157.330
C07036=1067.040,446.882,378.126,176.709,38.217,157.326
C07037=1067.031,446.638,378.176,176.697,38.202,157.322
C07038=1067.021,446.393,378.226,176.687,38.188,157.318
C07039=1067.011,446.148,378.276,176.677,38.173,157.314
C07040=1067.001,445.904,378.326,176.666,38.159,157.309
C07041=1066.991,445.659,378.376,176.656,38.144,157.305
C07042=1066.982,445.414,378.426,176.646,38.130,157.301
C07043=1066.972,445.170,378.475,176.635,38.116,157.297
C07044=1066.962,444.925,378.526,176.625,38.102,157.293
C07045=1066.952,444.680,378.576,176.615,38.088,157.289
C07046=1066.943,444.435,378.625,176.605,38.073,157.285
C07047=1066.933,444.191,378.675,176.595,38.059,157.281
C07048=1066.923,443.946,378.725,176.584,38.045,157.278
C07049=1066.914,443.701,378.775,176.574,38.031,157.274
C07050=1066.904,443.457,378.824,176.564,38.017,157.270
C07051=1066.894,443.212,378.874,176.554,38.003,157.266
C07052=1066.885,442.967,378.922,176.544,37.989,157.262
C07053=1066.875,442.707,378.975,176.534,37.974,157.258
C07054=1066.864,442.448,379.027,176.524,37.960,157.254
C07055=1066.854,442.189,379.080,176.512,37.946,157.250
C07056=1066.844,441.930,379.131,176.502,37.931,157.246
C07057=1066.834,441.685,379.180,176.492,37.918,157.242
C07058=1066.825,441.440,379.230,176.483,37.904,157.238
C07059=1066.815,441.196,379.279,176.473,37.890,157.234
C07060=1066.806,440.950,379.328,176.464,37.877,157.231
C07061=1066.797,440.705,379.377,176.455,37.864,157.227
C07062=1066.787,440.460,379.426,176.445,37.850,157.223
C07063=1066.778,440.215,379.474,176.435,37.837,157.220
C07064=1066.769,439.970,379.523,176.426,37.823,157.216
C07065=1066.759,439.725,379.572,176.416,37.810,157.212
C07066=1066.750,439.480,379.621,176.406,37.797,157.209
C07067=1066.741,439.235,379.669,176.398,37.783,157.205
C07068=1066.731,438.990,379.718,176.388,37.771,157.202
C07069=1066.722,438.745,379.767,176.379,37.757,157.198
C07070=1066.712,438.500,379.815,176.370,37.745,157.195
C07071=1066.702,438.255,379.864,176.361,37.731,157.191
C07072=1066.694,438.010,379.912,176.351,37.718,157.187
C07073=1066.685,437.765,379.960,176.342,37.706,157.184
C07074=1066.675,437.520,380.009,176.333,37.693,157.180
C07075=1066.666,437.275,380.056,176.324,37.680,157.177
C07076=1066.656,437.030,380.105,176.315,37.667,157.173
C07077=1066.647,436.785,380.153,176.306,37.654,157.170
C07078=1066.638,436.540,380.201,176.296,37.641,157.166
C07079=1066.629,436.294,380.249,176.288,37.629,157.163
C07080=1066.619,436.049,380.297,176.278,37.616,157.160
C07081=1066.610,435.805,380.345,176.270,37.604,157.156
C07082=1066.601,435.559,380.393,176.261,37.591,157.153
C07083=1066.592,435.314,380.440,176.252,37.579,157.149
C07084=1066.582,435.068,380.488,176.243,37.566,157.146
C07085=1066.574,434.824,380.536,176.235,37.554,157.143
C07086=1066.565,434.578,380.584,176.226,37.541,157.139
C07087=1066.556,434.333,380.631,176.217,37.529,157.136
C07088=1066.547,434.087,380.679,176.208,37.517,157.133
C07089=1066.538,433.842,380.727,176.200,37.504,157.130
C07090=1066.529,433.597,380.774,176.192,37.492,157.126
C07091=1066.519,433.352,380.822,176.182,37.480,157.123
C07092=1066.511,433.107,380.869,176.174,37.468,157.120
C07093=1066.502,432.862,380.917,176.165,37.455,157.116
C07094=1066.493,432.616,380.964,176.157,37.444,157.113
C07095=1066.484,432.371,381.011,176.149,37.432,157.110
C07096=1066.475,432.126,381.059,176.140,37.419,157.107
C07097=1066.466,431.880,381.106,176.132,37.407,157.104
C07098=1066.457,431.635,381.153,176.123,37.395,157.100
C07099=1066.448,431.389,381.200,176.115,37.383,157.097
C07100=1066.439,431.144,381.248,176.106,37.372,157.094
C07101=1066.431,430.899,381.294,176.098,37.360,157.091
C07102=1066.422,430.654,381.342,176.090,37.348,157.088
C07103=1066.414,430.409,381.388,176.082,37.336,157.085
C07104=1066.404,430.163,381.435,176.073,37.324,157.081
C07105=1066.395,429.917,381.482,176.065,37.313,157.078
C07106=1066.386,429.672,381.529,176.057,37.301,157.075
C07107=1066.378,429.427,381.576,176.049,37.289,157.072
C07108=1066.369,429.181,381.623,176.041,37.278,157.069
C07109=1066.358,428.865,381.683,176.031,37.263,157.065
C07110=1066.347,428.547,381.743,176.020,37.248,157.061
C07111=1066.335,428.231,381.803,176.009,37.233,157.057
C07112=1066.325,427.914,381.863,176.000,37.219,157.054
C07113=1066.315,427.668,381.909,175.992,37.207,157.051
C07114=1066.307,427.423,381.955,175.984,37.196,157.048
C07115=1066.298,427.177,382.002,175.976,37.185,157.045
C07116=1066.289,426.932,382.048,175.968,37.173,157.042
C07117=1066.281,426.686,382.094,175.961,37.162,157.039
C07118=1066.271,426.441,382.140,175.953,37.151,157.036
C07119=1066.263,426.195,382.187,175.945,37.140,157.033
C07120=1066.255,425.949,382.233,175.937,37.129,157.030
C07121=1066.246,425.705,382.279,175.929,37.118,157.027
C07122=1066.238,425.459,382.325,175.922,37.107,157.024
C07123=1066.229,425.213,382.370,175.914,37.096,157.022
C07124=1066.220,424.967,382.417,175.906,37.085,157.019
C07125=1066.211,424.721,382.463,175.898,37.074,157.016
C07126=1066.203,424.477,382.509,175.891,37.063,157.013
C07127=1066.194,424.231,382.554,175.883,37.052,157.010
C07128=1066.185,423.985,382.600,175.875,37.041,157.007
C07129=1066.177,423.739,382.646,175.868,37.030,157.004
C07130=1066.169,423.494,382.691,175.861,37.020,157.002
C07131=1066.160,423.248,382.738,175.853,37.009,156.999
C07132=1066.151,423.002,382.783,175.846,36.998,156.996
C07133=1066.143,422.757,382.829,175.838,36.987,156.993
C07134=1066.134,422.511,382.874,175.831,36.977,156.991
C07135=1066.127,422.266,382.920,175.823,36.966,156.988
C07136=1066.118,422.020,382.965,175.816,36.956,156.985
C07137=1066.110,421.774,383.011,175.809,36.945,156.982
C07138=1066.101,421.529,383.056,175.801,36.934,156.980
C07139=1066.093,421.282,383.101,175.794,36.924,156.977
C07140=1066.085,421.037,383.147,175.786,36.913,156.974
C07141=1066.076,420.791,383.192,175.780,36.903,156.972
C07142=1066.068,420.546,383.237,175.772,36.893,156.969
C07143=1066.060,420.299,383.282,175.765,36.882,156.966
C07144=1066.051,420.054,383.327,175.758,36.872,156.964
C07145=1066.043,419.807,383.372,175.751,36.861,156.961
C07146=1066.034,419.562,383.417,175.743,36.851,156.958
C07147=1066.026,419.316,383.462,175.736,36.841,156.956
C07148=1066.017,419.071,383.507,175.729,36.831,156.953
C07149=1066.010,418.825,383.552,175.722,36.821,156.951
C07150=1066.001,418.579,383.597,175.715,36.810,156.948
C07151=1065.993,418.333,383.642,175.708,36.800,156.945
C07152=1065.984,418.087,383.686,175.701,36.790,156.943
C07153=1065.976,417.842,383.731,175.694,36.780,156.940
C07154=1065.968,417.596,383.776,175.687,36.770,156.938
C07155=1065.959,417.349,383.820,175.680,36.760,156.935
C07156=1065.952,417.103,383.865,175.673,36.750,156.933
C07157=1065.943,416.858,383.910,175.666,36.740,156.930
C07158=1065.935,416.612,383.955,175.660,36.730,156.928
C07159=1065.927,416.366,383.999,175.653,36.720,156.925
C07160=1065.918,416.120,384.044,175.645,36.710,156.922
C07161=1065.910,415.874,384.088,175.639,36.701,156.920
C07162=1065.902,415.629,384.132,175.632,36.690,156.918
C07163=1065.894,415.383,384.177,175.625,36.681,156.915
C07164=1065.886,415.137,384.221,175.618,36.671,156.913
C07165=1065.877,414.840,384.275,175.610,36.659,156.910
C07166=1065.867,414.543,384.328,175.603,36.647,156.907
C07167=1065.857,414.246,384.381,175.594,36.636,156.904
C07168=1065.847,413.948,384.435,175.586,36.624,156.901
C07169=1065.838,413.702,384.479,175.579,36.614,156.898
C07170=1065.830,413.456,384.523,175.573,36.605,156.896
C07171=1065.822,413.210,384.567,175.566,36.596,156.894
C07172=1065.814,412.964,384.611,175.559,36.586,156.891
C07173=1065.806,412.718,384.654,175.553,36.577,156.889
C07174=1065.798,412.472,384.698,175.546,36.567,156.886
C07175=1065.790,412.226,384.742,175.540,36.558,156.884
C07176=1065.782,411.980,384.786,175.533,36.548,156.882
C07177=1065.774,411.734,384.830,175.527,36.539,156.880
C07178=1065.765,411.488,384.873,175.521,36.530,156.877
C07179=1065.758,411.242,384.917,175.513,36.520,156.875
C07180=1065.750,410.996,384.961,175.507,36.511,156.872
C07181=1065.741,410.750,385.004,175.501,36.502,156.870
C07182=1065.733,410.503,385.048,175.494,36.493,156.868
C07183=1065.725,410.258,385.092,175.488,36.483,156.866
C07184=1065.718,410.012,385.136,175.481,36.474,156.863
C07185=1065.710,409.766,385.179,175.475,36.465,156.861
C07186=1065.702,409.520,385.222,175.469,36.456,156.859
C07187=1065.694,409.273,385.266,175.462,36.447,156.857
C07188=1065.686,409.027,385.309,175.456,36.438,156.854
C07189=1065.678,408.781,385.353,175.450,36.428,156.852
C07190=1065.671,408.535,385.396,175.443,36.419,156.850
C07191=1065.662,408.289,385.439,175.437,36.410,156.847
C07192=1065.654,408.043,385.482,175.431,36.401,156.845
C07193=1065.647,407.796,385.526,175.425,36.392,156.843
C07194=1065.639,407.551,385.569,175.419,36.383,156.841
C07195=1065.631,407.305,385.612,175.413,36.374,156.839
C07196=1065.623,407.058,385.656,175.407,36.365,156.836
C07197=1065.615,406.813,385.699,175.401,36.357,156.834
C07198=1065.608,406.566,385.742,175.394,36.347,156.832
C07199=1065.600,406.320,385.785,175.388,36.339,156.830
C07200=1065.592,406.074,385.828,175.382,36.330,156.828
C07201=1065.585,405.827,385.871,175.376,36.321,156.825
C07202=1065.577,405.582,385.913,175.369,36.312,156.823
C07203=1065.569,405.336,385.957,175.364,36.303,156.821
C07204=1065.561,405.089,385.999,175.358,36.295,156.819
C07205=1065.554,404.843,386.043,175.352,36.286,156.817
C07206=1065.545,404.597,386.085,175.345,36.277,156.815
C07207=1065.538,404.351,386.128,175.339,36.269,156.813
C07208=1065.530,404.104,386.170,175.334,36.260,156.811
C07209=1065.523,403.858,386.212,175.328,36.252,156.808
C07210=1065.515,403.612,386.256,175.322,36.243,156.806
C07211=1065.507,403.366,386.298,175.316,36.234,156.804
C07212=1065.499,403.119,386.340,175.309,36.226,156.802
C07213=1065.492,402.874,386.384,175.304,36.217,156.800
C07214=1065.484,402.627,386.426,175.298,36.209,156.798
C07215=1065.476,402.381,386.468,175.292,36.200,156.796
C07216=1065.468,402.134,386.510,175.286,36.192,156.794
C07217=1065.461,401.888,386.553,175.281,36.183,156.792
C07218=1065.452,401.642,386.596,175.275,36.175,156.790
C07219=1065.445,401.396,386.638,175.269,36.167,156.788
C07220=1065.437,401.150,386.680,175.262,36.159,156.786
C07221=1065.428,400.856,386.730,175.256,36.148,156.783
C07222=1065.419,400.564,386.780,175.249,36.139,156.781
C07223=1065.410,400.271,386.830,175.243,36.129,156.779
C07224=1065.401,399.979,386.880,175.235,36.119,156.776
C07225=1065.393,399.733,386.922,175.230,36.111,156.774
C07226=1065.385,399.486,386.964,175.224,36.103,156.772
C07227=1065.378,399.239,387.006,175.218,36.094,156.770
C07228=1065.371,398.993,387.048,175.213,36.086,156.768
C07229=1065.363,398.747,387.090,175.207,36.078,156.766
C07230=1065.355,398.501,387.132,175.201,36.070,156.764
C07231=1065.348,398.254,387.174,175.196,36.061,156.762
C07232=1065.340,398.008,387.216,175.190,36.053,156.760
C07233=1065.332,397.762,387.258,175.185,36.046,156.759
C07234=1065.325,397.516,387.299,175.179,36.038,156.757
C07235=1065.318,397.270,387.341,175.173,36.029,156.755
C07236=1065.309,397.023,387.383,175.168,36.021,156.753
C07237=1065.302,396.776,387.424,175.162,36.014,156.751
C07238=1065.294,396.530,387.466,175.157,36.005,156.749
C07239=1065.287,396.284,387.507,175.151,35.998,156.747
C07240=1065.280,396.038,387.549,175.145,35.990,156.745
C07241=1065.272,395.791,387.591,175.140,35.982,156.743
C07242=1065.265,395.545,387.632,175.134,35.974,156.741
C07243=1065.257,395.299,387.674,175.129,35.966,156.740
C07244=1065.250,395.052,387.715,175.123,35.958,156.738
C07245=1065.243,394.805,387.756,175.118,35.950,156.736
C07246=1065.235,394.559,387.798,175.112,35.943,156.734
C07247=1065.228,394.313,387.839,175.107,35.935,156.732
C07248=1065.220,394.067,387.880,175.101,35.927,156.730
C07249=1065.212,393.821,387.922,175.096,35.919,156.728
C07250=1065.205,393.574,387.963,175.090,35.912,156.726
C07251=1065.198,393.327,388.004,175.085,35.904,156.725
C07252=1065.190,393.081,388.046,175.079,35.896,156.723
C07253=1065.182,392.835,388.086,175.074,35.889,156.721
C07254=1065.175,392.588,388.128,175.069,35.881,156.719
C07255=1065.168,392.341,388.169,175.064,35.873,156.717
C07256=1065.161,392.095,388.210,175.058,35.866,156.716
C07257=1065.153,391.848,388.251,175.053,35.858,156.714
C07258=1065.145,391.602,388.292,175.047,35.850,156.712
C07259=1065.139,391.356,388.333,175.042,35.843,156.710
C07260=1065.131,391.110,388.373,175.037,35.836,156.708
C07261=1065.123,390.863,388.415,175.031,35.828,156.707
C07262=1065.116,390.617,388.456,175.026,35.820,156.705
C07263=1065.108,390.370,388.496,175.021,35.813,156.703
C07264=1065.101,390.123,388.537,175.016,35.805,156.701
C07265=1065.094,389.877,388.577,175.010,35.798,156.700
C07266=1065.086,389.631,388.619,175.005,35.791,156.698
C07267=1065.078,389.385,388.659,175.000,35.783,156.696
C07268=1065.071,389.137,388.700,174.994,35.776,156.694
C07269=1065.063,388.891,388.740,174.989,35.769,156.693
C07270=1065.057,388.645,388.780,174.984,35.761,156.691
C07271=1065.049,388.398,388.821,174.979,35.754,156.689
C07272=1065.042,388.152,388.862,174.974,35.747,156.687
C07273=1065.034,387.905,388.902,174.968,35.739,156.686
C07274=1065.027,387.659,388.943,174.963,35.732,156.684
C07275=1065.019,387.412,388.983,174.958,35.725,156.682
C07276=1065.011,387.166,389.024,174.953,35.718,156.681
C07277=1065.003,386.889,389.068,174.947,35.710,156.679
C07278=1064.996,386.613,389.114,174.942,35.701,156.677
C07279=1064.988,386.337,389.159,174.936,35.694,156.675
C07280=1064.979,386.061,389.205,174.930,35.685,156.673
C07281=1064.972,385.814,389.245,174.925,35.678,156.672
